			// Base centrale non utilizzata della cavallina
			IF Supporto.Tipologia = CAVALLETTO    THEN
				B := Supporto.YDim - Supporto.DimBaseUtile - Supporto.DimBaseUtile;
				B2 := ( Supporto.YDim / 2 )-supporto.DimBaseUtile ;
				CorYIz := supporto.DimBaseUtile ;
				CorYDe := Supporto.YDim - supporto.DimBaseUtile ;
				BaseAlgulo := ( Supporto.YDim /2) - (Supporto.DimVertice /2)- supporto.DimBaseUtile;
			ELSE
				B := Supporto.YDim - Supporto.DimBaseUtile - Supporto.DimBaseUtile;
				B2 := ( Supporto.YDim / 2 )-supporto.DimBaseUtile ;
			END_IF
			
			//B := Supporto.YDim - Supporto.DimBaseUtile - Supporto.DimBaseUtile;
			//B2 := ( Supporto.YDim / 2 )-supporto.DimBaseUtile ;
			IF (B <= 0 ) THEN
				Errore := ErrBase;
				RETURN;
			END_IF
			
			IF (Supporto.DimBaseUtile <= 0 ) OR (Supporto.DimBaseUtile <= 0 ) THEN
				Errore := ErrLUtile;
			END_IF
			
			b1 := (B - Supporto.DimVertice) / 2;	// base del triangolo rettangolo dell'angolo alfa
			IF (b1 <= 0 ) THEN
				Errore := ErrBaseAlfa;
				RETURN;
			END_IF
			
			h1 := Supporto.HMAX - Supporto.ZDim; // Altezza del triangolo rettangolo dell'angolo alfa
			IF h1 <= 0 THEN
				Errore := ErrAltezzaAlfa;
				RETURN;
			END_IF
			
			(* calcolo angolo alfa dell'inclinazione appoggio della lastra *)
			AngoloAlfa_rad := ATAN( b1 / h1); // Angolo superiore appoggio cavallina (in radianti)
			AlgoloAlfa_gradi := rad_to_deg(AngoloAlfa_rad); 
			
			IF (AlgoloAlfa_gradi >= 90) THEN
				Errore := ErrAngolo;
				RETURN;
			END_IF
			
			(* Calcolo angolo beta dell'eventuale piano di appoggio inclinato della cavallina*)
			AngoloBeta_rad := ATAN( (Supporto.ZDim_Ext1 - Supporto.ZDim) / Supporto.DimBaseUtile); 	// Angolo del piano di appoggio inclinato della cavallina (in radianti)
			AngoloBeta_gradi := rad_to_deg(AngoloBeta_rad);					// Angolo del piano di appoggio inclinato della cavallina (in gradi)
			rad90 := deg_to_rad(90);
			
			IF (AlgoloAlfa_gradi < (AngoloBeta_gradi-1)) AND FALSE (*Quitar alarma pendiente base*) THEN
				Errore := ErrPendenzaBase;					// Angolo alfa deve essere maggiore dell'angolo beta
				RETURN;
			END_IF
			
			// Calcolo lo spessore di ogni singola lastra/falda depositata sul lato della cavallina
			Spessore_Lastra_Inclinata[1] := 0;
			FOR counter2:=2 TO MAXFORMINGSLAB/2 BY 1 DO
				Spessore_Lastra_Inclinata[counter2] := Materiale[TipoElementoDep[counter2-1]].ZDim / COS(AngoloAlfa_rad);
			END_FOR;
			
			// Calcola lo spessore complessivo fino al passo n delle lastre/falde depositate sul singolo lato della cavallina 
			//memset(ADR(Spessore_Lastra_Inclinata_Cumulato), 0 , SIZEOF(Spessore_Lastra_Inclinata_Cumulato));
			
			IF (Spessore_Lastra_Inclinata_Cumulato[2] = 0) THEN
				FOR counter2:=1 TO MAXFORMINGSLAB/2 BY 1 DO
					FOR counter1 := 1 TO counter2 BY 1 DO
						Spessore_Lastra_Inclinata_Cumulato[counter2] := Spessore_Lastra_Inclinata_Cumulato[counter2]+Spessore_Lastra_Inclinata[counter1];
					END_FOR
				END_FOR
			END_IF
			
			// Numero di possibili lastre sul singolo lato
			//FOR counter1:=1 TO MAXFORMINGSLAB/2 BY 1 DO
				//IF (OrdineDeposito[counter1] <> e_Tipo_Elemento_Da_Lavorare.NOT_DEFINED AND OrdineDeposito[counter1] <> TERMINATORE) AND 
				//	((Spessore_Lastra_Inclinata_Cumulato[counter1] >0) AND (Spessore_Lastra_Inclinata_Cumulato[counter1] < Supporto.DimBaseUtile)) THEN
				//		numeroLastre_int := counter1;
				//END_IF
				//IF (OrdineDeposito[counter1] <> e_Tipo_Elemento_Da_Lavorare.NOT_DEFINED AND OrdineDeposito[counter1] <> TERMINATORE) AND 
				//	(Spessore_Lastra_Inclinata_Cumulato[counter1] >= Supporto.DimBaseUtile) THEN
				//		Errore := ErrNumeroPezzi;	// il supervisore mi ha passato troppe lastre rispetto allo spazio utile
				//END_IF
			//END_FOR
			IF (Spessore_Lastra_Inclinata_Cumulato[numeroLastre_int] >= Supporto.DimBaseUtile*2) THEN
				Errore := ErrNumeroPezzi;	// il supervisore mi ha passato troppe lastre rispetto allo spazio utile
			END_IF
			
			// Calcolo lo spostamento del punto centrale e del punto esterno della singola lastra/falda rispetto al punto interno(iniziale) della medesima lastra/falda
			FOR counter2:=1 TO numeroLastre_int BY 1 DO
				Yd1[counter2] := Materiale[TipoElementoDep[counter2]].ZDim / 2 * COS (AngoloAlfa_rad);		// Spostamento Centro lastra da interno lastra in Y
				Zd1[counter2] := Materiale[TipoElementoDep[counter2]].ZDim / 2 * SIN (AngoloAlfa_rad);		// Spostamento Centro lastra da interno lastra in Z
				Yd2[counter2] := Materiale[TipoElementoDep[counter2]].ZDim  * COS (AngoloAlfa_rad);			// Spostamento esterno lastra da interno lastra in Y
				Zd2[counter2] := Materiale[TipoElementoDep[counter2]].ZDim  * SIN (AngoloAlfa_rad);			// Spostamento esterno lastra da interno lastra in Z
			END_FOR
			
			// Calcolo la proiezione mancante di ogni singola lastra/falda; Tramite CI posso calcolare lo spostamento Yd3,Zd3 dovuto al piano inclinato
			// dovuto all'angolo beta. Utilizzo il teorema dei seni per calcolare ogni CI da SLIC
			FOR counter1:=1 TO numeroLastre_int BY 1 DO
				CI[counter1] := (Spessore_Lastra_Inclinata_Cumulato[counter1] * SIN (AngoloBeta_rad) ) / SIN( rad90 + AngoloAlfa_rad - AngoloBeta_rad);
				Yd3[counter1] := -CI[counter1] * SIN(AngoloAlfa_rad);
				Zd3[counter1] := CI[counter1] * COS(AngoloAlfa_rad);
			END_FOR;
			
			// Quota Y e Z del punto di appoggio di ogni lastra sulla cavallina
			// Quota Y e Z del punto interno centrale di ogni lastra; corrisponde a YInternoLastra e ZInternoLastra
			NuPiezasLadoDx := 0 ;
			NuPiezasLadoSx := 0 ;
			FOR counter2:=1 TO numeroLastre_int BY 1 DO
				XInternoLastra[counter2] := Supporto.XDim/2;
				varEven := counter2 MOD 2;
				IF Supporto.Tipologia = CAVALLETTO    THEN
					CASE varEven OF
						0:	
								CASE TipoCalculo OF
								0:
									YCoordinataAppoggioLastra[counter2] := (B/2) + Spessore_Lastra_Inclinata_Cumulato[counter2] + Yd3[counter2];
								
								
								1: 
									NuPiezasLadoDx := NuPiezasLadoDx +1 ;
									YCoordinataAppoggioLastra[counter2] := (CorYDe) + Spessore_Lastra_Inclinata_Cumulato[NuPiezasLadoDx] + Yd3[NuPiezasLadoDx];
									
								END_CASE
						1:
							CASE TipoCalculo OF
								0:
									YCoordinataAppoggioLastra[counter2] := (B/2) + Spessore_Lastra_Inclinata_Cumulato[counter2] - Yd3[counter2];
								
								1:
									NuPiezasLadoSx := NuPiezasLadoSx + 1;
									YCoordinataAppoggioLastra[counter2] := (CorYIz) + Spessore_Lastra_Inclinata_Cumulato[NuPiezasLadoSx] - Yd3[NuPiezasLadoSx];
							END_CASE
					END_CASE
					
					
					ELSE
					YCoordinataAppoggioLastra[counter2] := (B/2) + Spessore_Lastra_Inclinata_Cumulato[counter2] + Yd3[counter2];
						
				END_IF
				//YCoordinataAppoggioLastra[counter2] := (*(B2) +*) Spessore_Lastra_Inclinata_Cumulato[counter2] + Yd3[counter2];
				YInternoLastra[counter2] := YCoordinataAppoggioLastra[counter2] - (Materiale[TipoElementoDep[counter2]].YDim / 2) * SIN (AngoloAlfa_rad);
				ZCoordinataAppoggioLastra[counter2] := Supporto.ZDim + Zd3[counter2];
				ZInternoLastra[counter2] := ZCoordinataAppoggioLastra[counter2] + (Materiale[TipoElementoDep[counter2]].YDim / 2) * COS (AngoloAlfa_rad); 
			END_FOR
	
			(* Calcolo delle coordinate X,Y,Z di ogni singola lastra/falda, centrale o esterno *)
			FOR counter2:=1 TO numeroLastre_int BY 1 DO
				XCentroLastra[counter2] := Supporto.XDim/2;
				YCentroLastra[counter2] := YInternoLastra[counter2] + Yd1[counter2];
				ZCentroLastra[counter2] := ZInternoLastra[counter2] + Zd1[counter2];
				
				XEsternoLastra[counter2] := Supporto.XDim/2;
				YEsternoLastra[counter2] := YInternoLastra[counter2] + Yd2[counter2];	
				ZEsternoLastra[counter2] := ZInternoLastra[counter2] + Zd2[counter2];
			END_FOR;
			
			(* Pulisco le uscite e setto a TERMINATORE tutti gli elementi di FormingSlab*)
			FOR counter1 := 1 TO MAXFORMINGSLAB DO
				FormingSlab.PElement[counter1].Typology := TERMINATORE;
			END_FOR
		//#########################aqui for	
		IF HabiCalTodasCordenadas THEN
				F_ini := 1 ;
				F_Fin := 4 ;
			ELSE
				F_ini := TipoOrdinamento ;
				F_Fin := TipoOrdinamento ;
		END_IF
		FOR CalForCavallete := F_ini TO F_Fin DO
			(* Calcolo delle coordinate X,Y,Z,J del punto finale sulla base del TipoRisultato *)
			CASE CalForCavallete OF
				(* Ordinamento alternato Dx-SX *)	
				1: 
					FOR counter2:=1 TO numeroLastre_int*2 BY 1 DO
						varEven := counter2 MOD 2;	
						CASE varEven OF
							0:	// Lato DX della cavallina
								XFinale[counter2] := Supporto.XDim/2 + Supporto.OFSDE_X180;
								CASE TipoRisultato OF
									1:	
										YFinale[counter2] := -YInternoLastra[(counter2+varEven)/2] + Supporto.OFSDE_Y180;
										ZFinale[counter2] := ZInternoLastra[(counter2+varEven)/2] + Supporto.OFSDE_Z180;
									2:	
										YFinale[counter2] := -YCentroLastra[(counter2+varEven)/2] + Supporto.OFSDE_Y180;
										ZFinale[counter2] := ZCentroLastra[(counter2+varEven)/2] + Supporto.OFSDE_Z180;
									3:	
										YFinale[counter2] := -YEsternoLastra[(counter2+varEven)/2] + Supporto.OFSDE_Y180;
										ZFinale[counter2] := ZEsternoLastra[(counter2+varEven)/2] + Supporto.OFSDE_Z180;
									4:	
										YFinale[counter2] := -YCoordinataAppoggioLastra[(counter2+varEven)/2] + Supporto.OFSDE_Y180;
										ZFinale[counter2] := ZEsternoLastra[(counter2+varEven)/2] + Supporto.OFSDE_Z180;
								END_CASE
								JFinale[counter2] := 180 - AlgoloAlfa_gradi + Supporto.OFSDE_J180; 
							1:	// Lato SX della cavallina
								XFinale[counter2] := Supporto.XDim/2 + Supporto.OFSDE_X0;
								CASE TipoRisultato OF
									1:	
										YFinale[counter2] := YInternoLastra[(counter2+varEven)/2] + Supporto.OFSDE_Y0;
										ZFinale[counter2] := ZInternoLastra[(counter2+varEven)/2] + Supporto.OFSDE_Z0;
									2:	
										YFinale[counter2] := YCentroLastra[(counter2+varEven)/2] + Supporto.OFSDE_Y0;
										ZFinale[counter2] := ZCentroLastra[(counter2+varEven)/2] + Supporto.OFSDE_Z0;
									3:	
										YFinale[counter2] := YEsternoLastra[(counter2+varEven)/2] + Supporto.OFSDE_Y0;
										ZFinale[counter2] := ZEsternoLastra[(counter2+varEven)/2] + Supporto.OFSDE_Z0;
									4:	
										YFinale[counter2] := YCoordinataAppoggioLastra[(counter2+varEven)/2] + Supporto.OFSDE_Y0;
										ZFinale[counter2] := ZEsternoLastra[(counter2+varEven)/2] + Supporto.OFSDE_Z0;
								END_CASE
								JFinale[counter2] := AlgoloAlfa_gradi + Supporto.OFSDE_J0;
						END_CASE
					END_FOR
					
				(* Ordinamento consecutivo prima un lato poi l'altro *)
				2:	
					FOR  CntLados :=  1 TO 2 BY 1 DO
						CASE CntLados OF 
							1:
								FOR counter2 :=1 TO numeroLastre_int BY 1 DO
										CoorFinaleLado_Pri0_Des180[counter2].LadoA.CoordenadaFinale_X := Supporto.XDim/2 + Supporto.OFSDE_X180;
									CASE TipoRisultato OF	
										1:	
											CoorFinaleLado_Pri0_Des180[counter2].LadoA.CoordenadaFinale_Y := YInternoLastra[counter2] + Supporto.OFSDE_Y0;
											CoorFinaleLado_Pri0_Des180[counter2].LadoA.CoordenadaFinale_Z := ZInternoLastra[counter2] + Supporto.OFSDE_Z0;
										2:	
											CoorFinaleLado_Pri0_Des180[counter2].LadoA.CoordenadaFinale_Y := YCentroLastra[counter2] + Supporto.OFSDE_Y0;
											CoorFinaleLado_Pri0_Des180[counter2].LadoA.CoordenadaFinale_Z := ZCentroLastra[counter2] + Supporto.OFSDE_Z0;
										3:	
											CoorFinaleLado_Pri0_Des180[counter2].LadoA.CoordenadaFinale_Y := YEsternoLastra[counter2] + Supporto.OFSDE_Y0;
											CoorFinaleLado_Pri0_Des180[counter2].LadoA.CoordenadaFinale_Z := ZEsternoLastra[counter2] + Supporto.OFSDE_Z0;
										4:	
											CoorFinaleLado_Pri0_Des180[counter2].LadoA.CoordenadaFinale_Y := YCoordinataAppoggioLastra[counter2] + Supporto.OFSDE_Y0;
											CoorFinaleLado_Pri0_Des180[counter2].LadoA.CoordenadaFinale_Z := ZEsternoLastra[counter2] + Supporto.OFSDE_Z0;
									END_CASE
									CoorFinaleLado_Pri0_Des180[counter2].LadoA.CoordenadaFinale_J := AlgoloAlfa_gradi + Supporto.OFSDE_J0;
								END_FOR
								2: 
									FOR counter2:=1 TO numeroLastre_int BY 1 DO
										
										CoorFinaleLado_Pri0_Des180[counter2].LadoA.CoordenadaFinale_X := Supporto.XDim/2 + Supporto.OFSDE_X180;
										CASE TipoRisultato OF
											1:	
												CoorFinaleLado_Pri0_Des180[counter2].LadoB.CoordenadaFinale_Y := -YInternoLastra[counter2] + Supporto.OFSDE_Y180;
												CoorFinaleLado_Pri0_Des180[counter2].LadoB.CoordenadaFinale_Z := ZInternoLastra[counter2] + Supporto.OFSDE_Z180;
											2:	
												CoorFinaleLado_Pri0_Des180[counter2].LadoB.CoordenadaFinale_Y := -YCentroLastra[counter2] + Supporto.OFSDE_Y180;
												CoorFinaleLado_Pri0_Des180[counter2].LadoB.CoordenadaFinale_Z := ZCentroLastra[counter2] + Supporto.OFSDE_Z180;
											3:	
												CoorFinaleLado_Pri0_Des180[counter2].LadoB.CoordenadaFinale_Y := -YEsternoLastra[counter2] + Supporto.OFSDE_Y180;
												//YFinale[counter2] := YCoordinataAppoggioLastra[counter2] ;
												CoorFinaleLado_Pri0_Des180[counter2].LadoB.CoordenadaFinale_Z := ZEsternoLastra[counter2] + Supporto.OFSDE_Z180;
											4:	
												CoorFinaleLado_Pri0_Des180[counter2].LadoB.CoordenadaFinale_Y := -YCoordinataAppoggioLastra[counter2] + Supporto.OFSDE_Y180;
												CoorFinaleLado_Pri0_Des180[counter2].LadoB.CoordenadaFinale_Z := ZEsternoLastra[counter2] + Supporto.OFSDE_Z180;
										END_CASE
										CoorFinaleLado_Pri0_Des180[counter2].LadoB.CoordenadaFinale_J := 180 - AlgoloAlfa_gradi + Supporto.OFSDE_J180; 
									END_FOR
													
							
							END_CASE
						END_FOR
						
							IF NOT HabiCalTodasCordenadas THEN 
								FOR counter2:=1 TO numeroLastre_int BY 1 DO
								IF counter2 <= numeroLastre_int/2 THEN // Lato DX della cavallina
									varEven := counter2 MOD 2;
									XFinale[counter2] := Supporto.XDim/2 + Supporto.OFSDE_X180;
									CASE TipoRisultato OF
										1:	
											YFinale[counter2] := -YInternoLastra[counter2] + Supporto.OFSDE_Y180;
											ZFinale[counter2] := ZInternoLastra[counter2] + Supporto.OFSDE_Z180;
										2:	
											YFinale[counter2] := -YCentroLastra[counter2] + Supporto.OFSDE_Y180;
											ZFinale[counter2] := ZCentroLastra[counter2] + Supporto.OFSDE_Z180;
										3:	
											YFinale[counter2] := -YEsternoLastra[counter2] + Supporto.OFSDE_Y180;
											ZFinale[counter2] := ZEsternoLastra[counter2] + Supporto.OFSDE_Z180;
										4:	
											YFinale[counter2] := -YCoordinataAppoggioLastra[counter2] + Supporto.OFSDE_Y180;
											ZFinale[counter2] :=  ZEsternoLastra[counter2] + Supporto.OFSDE_Z180;
									END_CASE
											JFinale[counter2] := 180 - AlgoloAlfa_gradi + Supporto.OFSDE_J180; 
								ELSE// Lato SX della cavallina
									XFinale[counter2] := Supporto.XDim/2 + Supporto.OFSDE_X0;
									CASE TipoRisultato OF
										1:	
											YFinale[counter2] := YInternoLastra[counter2-numeroLastre_int/2] + Supporto.OFSDE_Y0;
											ZFinale[counter2] := ZInternoLastra[counter2-numeroLastre_int/2] + Supporto.OFSDE_Z0;
										2:	
											YFinale[counter2] := YCentroLastra[counter2-numeroLastre_int/2] + Supporto.OFSDE_Y0;
											ZFinale[counter2] := ZCentroLastra[counter2-numeroLastre_int/2] + Supporto.OFSDE_Z0;
										3:	
											YFinale[counter2] := YEsternoLastra[counter2-numeroLastre_int/2] + Supporto.OFSDE_Y0;
											ZFinale[counter2] := ZEsternoLastra[counter2-numeroLastre_int/2] + Supporto.OFSDE_Z0;
										4:	
											YFinale[counter2] := YCoordinataAppoggioLastra[counter2-numeroLastre_int/2] + Supporto.OFSDE_Y0;
											ZFinale[counter2] := ZEsternoLastra[counter2-numeroLastre_int/2] + Supporto.OFSDE_Z0;
									END_CASE
									JFinale[counter2] := AlgoloAlfa_gradi + Supporto.OFSDE_J0;
								END_IF
							END_FOR
							END_IF
							
				(* Ordinamento consecutivo prima SOLO lato 0° *)
				3:
					FOR counter2:=1 TO numeroLastre_int BY 1 DO
						XFinaleLado_0Grados[counter2] := Supporto.XDim/2 + Supporto.OFSDE_X0;
						CASE TipoRisultato OF
							1:	
								YFinaleLado_0Grados[counter2] := YInternoLastra[counter2-numeroLastre_int/2] + Supporto.OFSDE_Y0;
								ZFinaleLado_0Grados[counter2] := ZInternoLastra[counter2-numeroLastre_int/2] + Supporto.OFSDE_Z0;
							2:	
								YFinaleLado_0Grados[counter2] := YCentroLastra[counter2-numeroLastre_int/2] + Supporto.OFSDE_Y0;
								ZFinaleLado_0Grados[counter2] := ZCentroLastra[counter2-numeroLastre_int/2] + Supporto.OFSDE_Z0;
							3:	
								YFinaleLado_0Grados[counter2] := YEsternoLastra[counter2-numeroLastre_int/2] + Supporto.OFSDE_Y0;
								ZFinaleLado_0Grados[counter2] := ZEsternoLastra[counter2-numeroLastre_int/2] + Supporto.OFSDE_Z0;
							4:	
								YFinaleLado_0Grados[counter2] := YCoordinataAppoggioLastra[counter2-numeroLastre_int/2] + Supporto.OFSDE_Y0;
								ZFinaleLado_0Grados[counter2] := ZEsternoLastra[counter2-numeroLastre_int/2] + Supporto.OFSDE_Z0;
						END_CASE
						JFinaleLado_0Grados[counter2] := AlgoloAlfa_gradi + Supporto.OFSDE_J0;
					END_FOR
					IF NOT HabiCalTodasCordenadas THEN 
						FOR counter2:=1 TO numeroLastre_int BY 1 DO
						XFinale[counter2] := Supporto.XDim/2 + Supporto.OFSDE_X0;
						CASE TipoRisultato OF
							1:	
								YFinale[counter2] := YInternoLastra[counter2-numeroLastre_int/2] + Supporto.OFSDE_Y0;
								ZFinale[counter2] := ZInternoLastra[counter2-numeroLastre_int/2] + Supporto.OFSDE_Z0;
							2:	
								YFinale[counter2] := YCentroLastra[counter2-numeroLastre_int/2] + Supporto.OFSDE_Y0;
								ZFinale[counter2] := ZCentroLastra[counter2-numeroLastre_int/2] + Supporto.OFSDE_Z0;
							3:	
								YFinale[counter2] := YEsternoLastra[counter2-numeroLastre_int/2] + Supporto.OFSDE_Y0;
								ZFinale[counter2] := ZEsternoLastra[counter2-numeroLastre_int/2] + Supporto.OFSDE_Z0;
							4:	
								YFinale[counter2] := YCoordinataAppoggioLastra[counter2-numeroLastre_int/2] + Supporto.OFSDE_Y0;
								ZFinale[counter2] := ZEsternoLastra[counter2-numeroLastre_int/2] + Supporto.OFSDE_Z0;
						END_CASE
						JFinale[counter2] := AlgoloAlfa_gradi + Supporto.OFSDE_J0;
					END_FOR
					END_IF
				(* Ordinamento consecutivo SOLO lato 180 *)
				4:
					FOR counter2:=1 TO numeroLastre_int BY 1 DO
						varEven := counter2 MOD 2;
						XFinaleLado_180Grados[counter2] := Supporto.XDim/2 + Supporto.OFSDE_X180;
						CASE TipoRisultato OF
							1:	
								YFinaleLado_180Grados[counter2] := -YInternoLastra[counter2] + Supporto.OFSDE_Y180;
								ZFinaleLado_180Grados[counter2] := 	ZInternoLastra[counter2] + Supporto.OFSDE_Z180;
							2:	
								YFinaleLado_180Grados[counter2] := -YCentroLastra[counter2] + Supporto.OFSDE_Y180;
								ZFinaleLado_180Grados[counter2] := ZCentroLastra[counter2] + Supporto.OFSDE_Z180;
							3:	
								YFinaleLado_180Grados[counter2] := -YEsternoLastra[counter2] + Supporto.OFSDE_Y180;
								//YFinale[counter2] := YCoordinataAppoggioLastra[counter2] ;
								ZFinaleLado_180Grados[counter2] := ZEsternoLastra[counter2] + Supporto.OFSDE_Z180;
							4:	
								YFinaleLado_180Grados[counter2] := -YCoordinataAppoggioLastra[counter2] + Supporto.OFSDE_Y180;
								ZFinaleLado_180Grados[counter2] := ZEsternoLastra[counter2] + Supporto.OFSDE_Z180;
						END_CASE
						JFinaleLado_180Grados[counter2] := 180 - AlgoloAlfa_gradi + Supporto.OFSDE_J180; 
					END_FOR
					IF NOT HabiCalTodasCordenadas THEN 
						FOR counter2:=1 TO numeroLastre_int BY 1 DO
						varEven := counter2 MOD 2;
						XFinale[counter2] := Supporto.XDim/2 + Supporto.OFSDE_X180;
						CASE TipoRisultato OF
							1:	
								YFinale[counter2] := -YInternoLastra[counter2] + Supporto.OFSDE_Y180;
								ZFinale[counter2] := ZInternoLastra[counter2] + Supporto.OFSDE_Z180;
							2:	
								YFinale[counter2] := -YCentroLastra[counter2] + Supporto.OFSDE_Y180;
								ZFinale[counter2] := ZCentroLastra[counter2] + Supporto.OFSDE_Z180;
							3:	
								YFinale[counter2] := -YEsternoLastra[counter2] + Supporto.OFSDE_Y180;
								//YFinale[counter2] := YCoordinataAppoggioLastra[counter2] ;
								ZFinale[counter2] := ZEsternoLastra[counter2] + Supporto.OFSDE_Z180;
							4:	
								YFinale[counter2] := -YCoordinataAppoggioLastra[counter2] + Supporto.OFSDE_Y180;
								ZFinale[counter2] := ZEsternoLastra[counter2] + Supporto.OFSDE_Z180;
						END_CASE
						JFinale[counter2] := 180 - AlgoloAlfa_gradi + Supporto.OFSDE_J180; 
					END_FOR
					END_IF
		
			5:
					;		
					
					
			END_CASE						
		END_FOR


			
			// Alimentazione della struttura FormingSlab
			FOR counter1:=1 TO MAXFORMINGSLAB DO// numeroLastre_int*2 BY 1 DO
				IF counter1 <= numeroLastre_int THEN
					FormingSlab.Enable := 1;										// Abilitato
					//FormingSlab.Code[1] := 1;
					FormingSlab.PElement[counter1].Typology 			:= OrdineDepositoSxDx[counter1];
					FormingSlab.PElement[counter1].X 					:= XFinale[counter1];
					FormingSlab.PElement[counter1].XDim 				:= Materiale[OrdineDepositoSxDx[counter1]].XDim;		// Dimensione X Lastra
					FormingSlab.PElement[counter1].Y 					:= YFinale[counter1];
					FormingSlab.PElement[counter1].YDim 				:= Materiale[OrdineDepositoSxDx[counter1]].YDim;		// Dimensione Y Lastra
					FormingSlab.PElement[counter1].Z 					:= ZFinale[counter1];
					FormingSlab.PElement[counter1].ZDim 				:= Materiale[OrdineDepositoSxDx[counter1]].ZDim;		// Dimensione Z Lastra
					FormingSlab.PElement[counter1].J 					:= JFinale[counter1];
					FormingSlab.PElement[counter1].CooCavallete 		:= CoorFinaleLado_Pri0_Des180[counter1] ;
				ELSE
					FormingSlab.PElement[counter1].Typology := OrdineDepositoSxDx[counter1];
					FormingSlab.PElement[counter1].X 		:= -1;
					FormingSlab.PElement[counter1].XDim 	:= -1;	
					FormingSlab.PElement[counter1].Y 		:= -1;
					FormingSlab.PElement[counter1].YDim 	:= -1;		
					FormingSlab.PElement[counter1].Z 		:= -1;
					FormingSlab.PElement[counter1].ZDim 	:= -1;	
					FormingSlab.PElement[counter1].J 		:= -1;
				END_IF
			END_FOR		
		

		INCLINATO_LATOSINGOLO:		// Tipo deposito inclinato singolo lato (Bundle)
			numeroLastre_int := 0;
			FOR counter1:=1 TO MAXFORMINGSLAB/2 BY 1 DO
				IF (TipoElementoDep[counter1] > 0) THEN
				numeroLastre_int := numeroLastre_int+1;
				END_IF;
			END_FOR
	
			(* Controlli dati coerenti --- DA FARE --- *)
						
			(* calcolo angolo alfa dell'inclinazione appoggio della lastra *)
			AngoloAlfa_rad := deg_to_rad(Supporto.AngoloAlfaBundle); // Angolo superiore appoggio cavallina (in radianti)
			AlgoloAlfa_gradi := Supporto.AngoloAlfaBundle; 
			
			
			(* Calcolo angolo beta dell'eventuale piano di appoggio inclinato della cavallina*)
			AngoloBeta_rad := AngoloAlfa_rad; 	// Angolo del piano di appoggio inclinato della cavallina (in radianti)
			AngoloBeta_gradi := AlgoloAlfa_gradi;					// Angolo del piano di appoggio inclinato della cavallina (in gradi)
	
			
			// Calcolo lo spessore di ogni singola lastra/falda depositata sul lato della cavallina
			Spessore_Lastra_Inclinata[1] := 0;
			FOR counter2:=2 TO MAXFORMINGSLAB/2 BY 1 DO
				Spessore_Lastra_Inclinata[counter2] := Materiale[TipoElementoDep[counter2-1]].ZDim / COS(AngoloAlfa_rad);
			END_FOR;
			
			// Calcola lo spessore complessivo fino al passo n delle lastre/falde depositate sul singolo lato della cavallina 
			//memset(ADR(Spessore_Lastra_Inclinata_Cumulato), 0 , SIZEOF(Spessore_Lastra_Inclinata_Cumulato));
			
			IF (Spessore_Lastra_Inclinata_Cumulato[2] = 0) THEN
				FOR counter2:=1 TO MAXFORMINGSLAB/2 BY 1 DO
					FOR counter1 := 1 TO counter2 BY 1 DO
						Spessore_Lastra_Inclinata_Cumulato[counter2] := Spessore_Lastra_Inclinata_Cumulato[counter2]+Spessore_Lastra_Inclinata[counter1];
					END_FOR
				END_FOR
			END_IF
			
			// Numero di possibili lastre sul singolo lato
			FOR counter1:=1 TO MAXFORMINGSLAB/2 BY 1 DO
				IF (TipoElementoDep[counter1] > 0) AND ((Spessore_Lastra_Inclinata_Cumulato[counter1] >0) AND (Spessore_Lastra_Inclinata_Cumulato[counter1] < Supporto.DimBaseUtile)) THEN
					numeroLastre_int := counter1;
				END_IF
				IF (Spessore_Lastra_Inclinata_Cumulato[counter1] >= Supporto.DimBaseUtile) THEN
					Errore := ErrNumeroPezzi;	// il supervisore mi ha passato troppe lastre rispetto allo spazio utile
				END_IF
			END_FOR
			
			// Calcolo lo spostamento del punto centrale e del punto esterno della singola lastra/falda rispetto al punto interno(iniziale) della medesima lastra/falda
			FOR counter2:=1 TO numeroLastre_int BY 1 DO
				Yd1[counter2] := Materiale[TipoElementoDep[counter2]].ZDim / 2 * COS (AngoloAlfa_rad);		// Spostamento Centro lastra da interno lastra in Y
				Zd1[counter2] := Materiale[TipoElementoDep[counter2]].ZDim / 2 * SIN (AngoloAlfa_rad);		// Spostamento Centro lastra da interno lastra in Z
				Yd2[counter2] := Materiale[TipoElementoDep[counter2]].ZDim  * COS (AngoloAlfa_rad);			// Spostamento esterno lastra da interno lastra in Y
				Zd2[counter2] := Materiale[TipoElementoDep[counter2]].ZDim  * SIN (AngoloAlfa_rad);			// Spostamento esterno lastra da interno lastra in Z
			END_FOR
			
			// Calcolo la proiezione mancante di ogni singola lastra/falda; Tramite CI posso calcolare lo spostamento Yd3,Zd3 dovuto al piano inclinato
			// dovuto all'angolo beta. Utilizzo il teorema dei seni per calcolare ogni CI da SLIC
			FOR counter1:=1 TO numeroLastre_int BY 1 DO
				CI[counter1] := (Spessore_Lastra_Inclinata_Cumulato[counter1] * SIN (AngoloBeta_rad));
				Yd3[counter1] := -CI[counter1] * SIN(AngoloAlfa_rad);
				Zd3[counter1] := CI[counter1] * COS(AngoloAlfa_rad);
			END_FOR;
			
			// Quota Y e Z del punto di appoggio di ogni lastra sulla cavallina
			// Quota Y e Z del punto interno centrale di ogni lastra; corrisponde a YInternoLastra e ZInternoLastra
			FOR counter2:=1 TO numeroLastre_int BY 1 DO
				XInternoLastra[counter2] := Supporto.XDim/2;
				YCoordinataAppoggioLastra[counter2] := Spessore_Lastra_Inclinata_Cumulato[counter2] + Yd3[counter2];
				YInternoLastra[counter2] := YCoordinataAppoggioLastra[counter2] - (Materiale[TipoElementoDep[counter2]].YDim / 2) * SIN (AngoloAlfa_rad);
				ZCoordinataAppoggioLastra[counter2] := Supporto.ZDim + Zd3[counter2];
				ZInternoLastra[counter2] := ZCoordinataAppoggioLastra[counter2] + (Materiale[TipoElementoDep[counter2]].YDim / 2) * COS (AngoloAlfa_rad); 
			END_FOR
	
			(* Calcolo delle coordinate X,Y,Z di ogni singola lastra/falda, centrale o esterno *)
			FOR counter2:=1 TO numeroLastre_int BY 1 DO
				XCentroLastra[counter2] := Supporto.XDim/2;
				YCentroLastra[counter2] := YInternoLastra[counter2] + Yd1[counter2];
				ZCentroLastra[counter2] := ZInternoLastra[counter2] + Zd1[counter2];
				
				XEsternoLastra[counter2] := Supporto.XDim/2;
				YEsternoLastra[counter2] := YInternoLastra[counter2] + Yd2[counter2];	
				ZEsternoLastra[counter2] := ZInternoLastra[counter2] + Zd2[counter2];
			END_FOR;
			
			(* Pulisco le uscite e setto a TERMINATORE tutti gli elementi di FormingSlab*)
			//memset(ADR(XFinale),0,SIZEOF(XFinale));memset(ADR(YFinale),0,SIZEOF(XFinale));memset(ADR(ZFinale),0,SIZEOF(XFinale));memset(ADR(JFinale),0,SIZEOF(XFinale));
			//memset(ADR(FormingSlab),0,SIZEOF(FormingSlab));
			FOR counter1 := 1 TO MAXFORMINGSLAB DO
				FormingSlab.PElement[counter1].Typology := TERMINATORE;
			END_FOR
			
			(* Calcolo delle coordinate X,Y,Z,J del punto finale sulla base del TipoRisultato *)
			FOR counter2:=1 TO numeroLastre_int BY 1 DO
				CASE supporto.LatoDeposito OF
					180:		// Lato DX della cavallina
						XFinale[counter2] := Supporto.XDim/2 + Supporto.OFSDE_X180;
						CASE TipoRisultato OF
							1:	
								YFinale[counter2] := -YInternoLastra[counter2] + Supporto.OFSDE_Y180;
								ZFinale[counter2] := ZInternoLastra[counter2] + Supporto.OFSDE_Z180;
							2:	
								YFinale[counter2] := -YCentroLastra[counter2] + Supporto.OFSDE_Y180;
								ZFinale[counter2] := ZCentroLastra[counter2] + Supporto.OFSDE_Z180;
							3:	
								YFinale[counter2] := -YEsternoLastra[counter2] + Supporto.OFSDE_Y180;
								ZFinale[counter2] := ZEsternoLastra[counter2] + Supporto.OFSDE_Z180;
						END_CASE
						JFinale[counter2] := 180 - AlgoloAlfa_gradi + Supporto.OFSDE_J180; 
					0:	// Lato SX della cavallina
						XFinale[counter2] := Supporto.XDim/2 + Supporto.OFSDE_X0;
						CASE TipoRisultato OF
							1:	
								YFinale[counter2] := YInternoLastra[counter2] + Supporto.OFSDE_Y0;
								ZFinale[counter2] := ZInternoLastra[counter2] + Supporto.OFSDE_Z0;
							2:	
								YFinale[counter2] := YCentroLastra[counter2] + Supporto.OFSDE_Y0;
								ZFinale[counter2] := ZCentroLastra[counter2] + Supporto.OFSDE_Z0;
							3:	
								YFinale[counter2] := YEsternoLastra[counter2] + Supporto.OFSDE_Y0;
								ZFinale[counter2] := ZEsternoLastra[counter2] + Supporto.OFSDE_Z0;
						END_CASE
						JFinale[counter2] := AlgoloAlfa_gradi + Supporto.OFSDE_J0;
				END_CASE

				
				// Alimentazione della struttura FormingSlab
				FOR counter1:=1 TO numeroLastre_int BY 1 DO
					FormingSlab.Enable := 1;										// Abilitato
					FormingSlab.Code[1] := 1;
					FormingSlab.PElement[counter1].Typology := Materiale[OrdineDepositoSxDx[counter1]].Typology;
					FormingSlab.PElement[counter1].X := XFinale[counter1];
					FormingSlab.PElement[counter1].XDim := Materiale[OrdineDepositoSxDx[counter1]].XDim;		// Dimensione X Lastra
					FormingSlab.PElement[counter1].Y := YFinale[counter1];
					FormingSlab.PElement[counter1].YDim := Materiale[OrdineDepositoSxDx[counter1]].YDim;		// Dimensione Y Lastra
					FormingSlab.PElement[counter1].Z := ZFinale[counter1];
					FormingSlab.PElement[counter1].ZDim := Materiale[OrdineDepositoSxDx[counter1]].ZDim;		// Dimensione Z Lastra
					FormingSlab.PElement[counter1].J := JFinale[counter1];
				END_FOR		
			END_FOR;	
	END_CASE


	// Salvataggio su file della Formatura 
	{region "Salvataggio File Formatura"}
	P_TextModeWrite.database[0,0] := 'X Finale';
	P_TextModeWrite.database[0,1] := 'Y Finale';
	P_TextModeWrite.database[0,2] := 'Z Finale';
	P_TextModeWrite.database[0,3] := 'J Finale';
	CASE TipoDeposito OF
		ORIZZONTALE :	
			P_TextModeWrite.database[0,4] := 'ORIZZONTALE';
			P_TextModeWrite.database[0,5] := UINT_TO_STRING(numeroLastre_int);
		INCLINATO : 
			P_TextModeWrite.database[0,4] := 'INCLINATO';
			P_TextModeWrite.database[0,5] := UINT_TO_STRING(numeroLastre_int*2);
		INCLINATO_LATOSINGOLO :
			P_TextModeWrite.database[0,4] := 'INCLINATO_LATOSINGOLO';
			P_TextModeWrite.database[0,5] := UINT_TO_STRING(numeroLastre_int);	  
	END_CASE
	CASE TipoRisultato OF
		1:	P_TextModeWrite.database[0,6] := 'PUNTO INTERNO';
		2:	P_TextModeWrite.database[0,6] := 'PUNTO CENTRALE';
		3:	P_TextModeWrite.database[0,6] := 'PUNTO ESTERNO';
	END_CASE
	
	FOR counter1 :=1 TO MAXFORMINGSLAB DO
		P_TextModeWrite.database[counter1,0] := LREAL_TO_STRING(XFinale[counter1]);
		P_TextModeWrite.database[counter1,1] := LREAL_TO_STRING(YFinale[counter1]);
		P_TextModeWrite.database[counter1,2] := LREAL_TO_STRING(ZFinale[counter1]);
		P_TextModeWrite.database[counter1,3] := LREAL_TO_STRING(JFinale[counter1]);
	END_FOR
	
	CASE TipoDeposito OF	// Numero di righe da scrivere sul file a seconda che sia CASSA o CAVALLINA
		ORIZZONTALE :	
			P_TextModeWrite.num_Row := numeroLastre_int;
		INCLINATO : 
			P_TextModeWrite.num_Row := numeroLastre_int * 2;
		INCLINATO_LATOSINGOLO : 
			P_TextModeWrite.num_Row := numeroLastre_int;
	END_CASE
	
	{endregion}
	CalcolaFormaturaDone := TRUE;	
	P_TextModeWrite.bWrite := TRUE; //Scrivo log per calcoli
ELSIF NOT CalcolaFormatura AND CalcolaFormaturaDone THEN
	CalcolaFormaturaDone := FALSE;
END_IF

//chiamata fb per log calcoli	
//___________P_TextModeWrite();
IF P_TextModeWrite.bWriteDone AND P_TextModeWrite.bWrite THEN
	P_TextModeWrite.bWrite := FALSE; 
END_IF

END_FUNCTION_BLOCK

// ---- POUs/TFPalletizerData_Lastre/Formatura/FuncionesFormacionParaquitar/Calcolo_Formatura_Completa_Back.TcPOU
FUNCTION_BLOCK Calcolo_Formatura_Completa_Back
VAR_INPUT
	
	Supporto : TFMachinePalletizer_Pallet;
	
	//Materiale : ARRAY [0..MAXTYPE_SLABLAYER] OF Type_SlabLayer;	// Tipo di materiale, Lastra, Falda e dimensioni
	Materiale 		: ARRAY [0..MAXTYPE_SLABLAYER] OF TFMachinePalletizer_PlaceElement;	// Tipo di materiale, Lastra, Falda e dimensioni
	TipoElementoDep 	: ARRAY [1..MAXFORMINGSLAB] OF e_Tipo_Elemento_Da_Lavorare;	// Tipologia del n-esimo elemento di Materiale da depositare (Lstra-falda-terminatore)
	
	TipoRisultato 		: UINT := 3;// Punto utilizzato per coordinate finali di deposito lastra/falda, 1 interno, 2 centro, 3 esterno(default)
	TipoOrdinamento 	: UINT := 1;//Tipologia di ordinamento in deposito 1= alternato (lastra DX-Lastra SX), 2 = consecutivo(prima un lato, poi l'altro lato), 3 = solo lato 0°, 4 = solo lato 180°
	NumeroElementiDaDepositare : UINT;

	PulisciMemoria : BOOL;
	CalcolaFormatura : BOOL;
END_VAR

VAR_OUTPUT
	(* Variabili di uscita della posizione finale del punto di deposito della lastra/falda *)
	XFinale : ARRAY [1..MAXFORMINGSLAB] OF LREAL;		// Coordinata X punto finale n-esima lastra/falda depositata
	YFinale : ARRAY [1..MAXFORMINGSLAB] OF LREAL;		// Coordinata Y punto finale n-esima lastra/falda depositata
	ZFinale : ARRAY [1..MAXFORMINGSLAB] OF LREAL;		// Coordinata Z punto finale n-esima lastra/falda depositata
	JFinale : ARRAY [1..MAXFORMINGSLAB] OF LREAL;		// Coordinata J punto finale n-esima lastra/falda depositata
	
	FormingSlab 			: TFMachinePalletizer_FormingForSlab;
	PulisciMemoriaDone		: BOOL;
	CalcolaFormaturaDone 	: BOOL;
	Errore 					: UINT;
END_VAR
VAR
	TipoDeposito : e_TipologiaDeposito;				// ORIZZONTALE O INCLINATO
	OrdineDepositoSxDx : ARRAY [1..MAXFORMINGSLAB] OF e_Tipo_Elemento_Da_Lavorare;	// Ordine deposito materiale per i due lati, sx e dx (considero di avere il medesimo ordine di deposito dai due lati) (CAVALLINA-INCLINATO)
	
	Spessore_Lastra_Inclinata : ARRAY [1..MAXFORMINGSLAB/2] OF LREAL;				// Occupazione in larghezza della singola lastra (CAVALLINA-INCLINATO)
	Spessore_Lastra_Inclinata_Cumulato : ARRAY [1..MAXFORMINGSLAB/2] OF LREAL;	// Occupazione in larghezza delle nlastre lastre cumulate (CAVALLINA)
	Spessore_Lastra : ARRAY [1..MAXFORMINGSLAB] OF LREAL;							// Occupazione in altezza della singola lastra (CASSA-ORIZZONTALE)
	Spessore_Lastra_Cumulato : ARRAY [1..MAXFORMINGSLAB] OF LREAL;					// Occupazione in altezza delle nlastre lastre cumulate (CASSA-ORIZZONTALE)
	
	YCoordinataAppoggioLastra :  ARRAY [1..MAXFORMINGSLAB/2] OF LREAL;		// Coordinata Y del punto di appoggio della lastra sulla base della cavallina  (CAVALLINA-INCLINATO)
	ZCoordinataAppoggioLastra :  ARRAY [1..MAXFORMINGSLAB/2] OF LREAL;		// Coordinata Z del punto di appoggio della lastra sulla base della cavallina  (CAVALLINA-INCLINATO)
	
	B 	: LREAL;	// Base della cavallina (include i due lati)  (CAVALLINA-INCLINATO)
	B2	: LREAL;	// Base della cavallina (include i due lati)  (CAVALLINA-INCLINATO)
	CorYIz  : LREAL;
	CorYDe : LREAL;
	BaseAlgulo : LREAL ;
	b1 : LREAL;	// base del triangolo rettangolo dell'angolo alfa  (CAVALLINA-INCLINATO)
	h1 : LREAL; // altezza del triangolo rettangolo dell'angolo alfa  (CAVALLINA-INCLINATO)
	Yd1 : ARRAY [1..MAXFORMINGSLAB/2] OF LREAL;	// Spostamento Centro lastra da inizio lastra in Y  (CAVALLINA-INCLINATO)
	Zd1 : ARRAY [1..MAXFORMINGSLAB/2] OF LREAL;	// Spostamento Centro lastra da inizio lastra in Z  (CAVALLINA-INCLINATO)
	Yd2 : ARRAY [1..MAXFORMINGSLAB/2] OF LREAL;	// Spostamento Esterno lastra da inizio lastra in Y  (CAVALLINA-INCLINATO)
	Zd2 : ARRAY [1..MAXFORMINGSLAB/2] OF LREAL;	// Spostamento Esterno lastra da inizio lastra in Z  (CAVALLINA-INCLINATOCAVALLINA)
	Yd3 : ARRAY [1..MAXFORMINGSLAB/2] OF LREAL;	// Spostamento Y dovuto al lato inclinato base appoggio  (CAVALLINA-INCLINATO)
	Zd3 : ARRAY [1..MAXFORMINGSLAB/2] OF LREAL;	// Spostamento Z dovuto al lato inclinato base appoggio  (CAVALLINA-INCLINATO)
	CI : ARRAY [1..MAXFORMINGSLAB/2] OF LREAL;	// Proiezione mancante della lastra dovuta al piano inclinato (CI) - Valorizzata solo se Beta >0  (CAVALLINA-INCLINATO)
	rad90 : LREAL;		// 90° in radianti
	
	(* Angoli piani appoggio lastre, laterale (alfa) e base (beta) cavallina *)
	AngoloAlfa_rad : LREAL;		// Angolo superiore laterale appoggio della lastra (in radianti)  (CAVALLINA-INCLINATO)
	AlgoloAlfa_gradi : LREAL; 	// Angolo superiore laterale appoggio della lastra (in gradi)  (CAVALLINA-INCLINATO)
	AngoloBeta_rad : LREAL;		// Angolo del piano inclinato di appoggio della lastra in radianti  (CAVALLINA-INCLINATO)
	AngoloBeta_gradi : LREAL; 	// Angolo del piano inclinato di appoggio della lastra in gradi  (CAVALLINA-INCLINATO)
	
	QuotaYinizioLastra : ARRAY [1..MAXFORMINGSLAB] OF LREAL;	// Quota Y inizio prima lastra  (CAVALLINA-INCLINATO)
	QuotaZinizioLastra : ARRAY [1..MAXFORMINGSLAB] OF LREAL;	// Quota Z inizio prima lastra  (CAVALLINA-INCLINATO)
	numeroLastre_int : UINT;									// Numero lastre per lato cavallina considerando la dimensione L_Utile1 (int)  (CAVALLINA-CASSA)
	
	(* Variabili di supporto *)
	counter1: UINT := 0;	// contatore per ciclo creazione formatura
	counter2: UINT := 0;	// contatore per ciclo creazione formatura
	varEven : UINT := 0;	// Pari o dispari per lato destro (dispari) o lato sinistro (pari) cavallina
	
	(* Variabili di uscita della posizione del punto interno, centrale ed esterno della lastra *)
	XInternoLastra : ARRAY [1..MAXFORMINGSLAB] OF LREAL;		// Coordinata X punto interno n-esima lastra depositata  (CAVALLINA-CASSA)
	YInternoLastra : ARRAY [1..MAXFORMINGSLAB] OF LREAL;		// Coordinata Y punto interno n-esima lastra depositata  (CAVALLINA-CASSA)
	ZInternoLastra : ARRAY [1..MAXFORMINGSLAB] OF LREAL;		// Coordinata Z punto interno n-esima lastra depositata  (CAVALLINA-CASSA)
	XCentroLastra  : ARRAY [1..MAXFORMINGSLAB] OF LREAL;		// Coordinata X punto centrale n-esima lastra depositata  (CAVALLINA-CASSA)
	YCentroLastra  : ARRAY [1..MAXFORMINGSLAB] OF LREAL;		// Coordinata Y punto centrale n-esima lastra depositata  (CAVALLINA-CASSA)
	ZCentroLastra  : ARRAY [1..MAXFORMINGSLAB] OF LREAL;		// Coordinata Z punto centrale n-esima lastra depositata  (CAVALLINA-CASSA)
	XEsternoLastra : ARRAY [1..MAXFORMINGSLAB] OF LREAL;		// Coordinata X punto esterno n-esima lastra depositata  (CAVALLINA-CASSA)
	YEsternoLastra : ARRAY [1..MAXFORMINGSLAB] OF LREAL;		// Coordinata Y punto esterno n-esima lastra depositata  (CAVALLINA-CASSA)
	ZEsternoLastra : ARRAY [1..MAXFORMINGSLAB] OF LREAL;		// Coordinata Z punto esterno n-esima lastra depositata  (CAVALLINA-CASSA)

	P_TextModeWrite : P_TextModeWrite;
	MemoriaInizializzata : BOOL;
END_VAR

VAR CONSTANT
END_VAR

// Pulisco le variabili interne e le variabili di uscita del FB
IF PulisciMemoria AND NOT PulisciMemoriaDone THEN		// Pulizia delle variabili locali e di uscita
	memset(ADR(XFinale), 0 , SIZEOF(XFinale));memset(ADR(YFinale), 0 , SIZEOF(YFinale));memset(ADR(ZFinale), 0 , SIZEOF(ZFinale));memset(ADR(JFinale), 0 , SIZEOF(JFinale));
	memset(ADR(FormingSlab), 0 , SIZEOF(FormingSlab));
	memset(ADR(Errore), 0 , SIZEOF(Errore));
	memset(ADR(OrdineDepositoSxDx), 0 , SIZEOF(OrdineDepositoSxDx));
	memset(ADR(Spessore_Lastra_Inclinata), 0 , SIZEOF(Spessore_Lastra_Inclinata));memset(ADR(Spessore_Lastra_Inclinata_Cumulato), 0 , SIZEOF(Spessore_Lastra_Inclinata_Cumulato));
	memset(ADR(Spessore_Lastra), 0 , SIZEOF(Spessore_Lastra));memset(ADR(Spessore_Lastra_Cumulato), 0 , SIZEOF(Spessore_Lastra_Cumulato));
	memset(ADR(YCoordinataAppoggioLastra), 0 , SIZEOF(YCoordinataAppoggioLastra));memset(ADR(ZCoordinataAppoggioLastra), 0 , SIZEOF(ZCoordinataAppoggioLastra));
	memset(ADR(B), 0 , SIZEOF(B));memset(ADR(b1), 0 , SIZEOF(b1));memset(ADR(h1), 0 , SIZEOF(h1));
	memset(ADR(Yd1), 0 , SIZEOF(Yd1));memset(ADR(Zd1), 0 , SIZEOF(Zd1));
	memset(ADR(Yd2), 0 , SIZEOF(Yd2));memset(ADR(Zd2), 0 , SIZEOF(Zd2));
	memset(ADR(Yd3), 0 , SIZEOF(Yd3));memset(ADR(Zd3), 0 , SIZEOF(Zd3));
	memset(ADR(CI), 0 , SIZEOF(CI));
	memset(ADR(AngoloAlfa_rad), 0 , SIZEOF(AngoloAlfa_rad));memset(ADR(AngoloBeta_rad), 0 , SIZEOF(AngoloBeta_rad));
	memset(ADR(QuotaYinizioLastra), 0 , SIZEOF(QuotaYinizioLastra));memset(ADR(QuotaZinizioLastra), 0 , SIZEOF(QuotaZinizioLastra));
	memset(ADR(numeroLastre_int), 0 , SIZEOF(numeroLastre_int));
	memset(ADR(XInternoLastra), 0 , SIZEOF(XInternoLastra));memset(ADR(YInternoLastra), 0 , SIZEOF(YInternoLastra));memset(ADR(ZInternoLastra), 0 , SIZEOF(ZInternoLastra));
	memset(ADR(XCentroLastra), 0 , SIZEOF(XCentroLastra));memset(ADR(YCentroLastra), 0 , SIZEOF(YCentroLastra));memset(ADR(ZCentroLastra), 0 , SIZEOF(ZCentroLastra));
	memset(ADR(XEsternoLastra), 0 , SIZEOF(XEsternoLastra));memset(ADR(YEsternoLastra), 0 , SIZEOF(YEsternoLastra));memset(ADR(ZEsternoLastra), 0 , SIZEOF(ZEsternoLastra));
	memset(ADR(Supporto), 0 , SIZEOF(Supporto));
	memset(ADR(Materiale), 0 , SIZEOF(Materiale));
	memset(ADR(TipoElementoDep), 99 , SIZEOF(TipoElementoDep));
	Errore := 0;
	PulisciMemoriaDone := TRUE;
	MemoriaInizializzata := TRUE;
ELSIF NOT PulisciMemoria AND PulisciMemoriaDone THEN
	PulisciMemoriaDone := FALSE;
END_IF

// Calcolo la Formatura, tipo Cassa o Cavallina e salvo su file i risultati ottenuti
IF CalcolaFormatura AND NOT CalcolaFormaturaDone AND MemoriaInizializzata THEN
	// Pulisco le variabili interne e le variabili di uscita del FB
	memset(ADR(XFinale), 0 , SIZEOF(XFinale));memset(ADR(YFinale), 0 , SIZEOF(YFinale));memset(ADR(ZFinale), 0 , SIZEOF(ZFinale));memset(ADR(JFinale), 0 , SIZEOF(JFinale));
	memset(ADR(FormingSlab), 0 , SIZEOF(FormingSlab));
	memset(ADR(Errore), 0 , SIZEOF(Errore));
	memset(ADR(OrdineDepositoSxDx), 0 , SIZEOF(OrdineDepositoSxDx));
	memset(ADR(Spessore_Lastra_Inclinata), 0 , SIZEOF(Spessore_Lastra_Inclinata));memset(ADR(Spessore_Lastra_Inclinata_Cumulato), 0 , SIZEOF(Spessore_Lastra_Inclinata_Cumulato));
	memset(ADR(Spessore_Lastra), 0 , SIZEOF(Spessore_Lastra));memset(ADR(Spessore_Lastra_Cumulato), 0 , SIZEOF(Spessore_Lastra_Cumulato));
	memset(ADR(YCoordinataAppoggioLastra), 0 , SIZEOF(YCoordinataAppoggioLastra));memset(ADR(ZCoordinataAppoggioLastra), 0 , SIZEOF(ZCoordinataAppoggioLastra));
	memset(ADR(B), 0 , SIZEOF(B));memset(ADR(b1), 0 , SIZEOF(b1));memset(ADR(h1), 0 , SIZEOF(h1));
	memset(ADR(Yd1), 0 , SIZEOF(Yd1));memset(ADR(Zd1), 0 , SIZEOF(Zd1));
	memset(ADR(Yd2), 0 , SIZEOF(Yd2));memset(ADR(Zd2), 0 , SIZEOF(Zd2));
	memset(ADR(Yd3), 0 , SIZEOF(Yd3));memset(ADR(Zd3), 0 , SIZEOF(Zd3));
	memset(ADR(CI), 0 , SIZEOF(CI));
	memset(ADR(AngoloAlfa_rad), 0 , SIZEOF(AngoloAlfa_rad));memset(ADR(AngoloBeta_rad), 0 , SIZEOF(AngoloBeta_rad));
	memset(ADR(QuotaYinizioLastra), 0 , SIZEOF(QuotaYinizioLastra));memset(ADR(QuotaZinizioLastra), 0 , SIZEOF(QuotaZinizioLastra));
	memset(ADR(numeroLastre_int), 0 , SIZEOF(numeroLastre_int));
	memset(ADR(XInternoLastra), 0 , SIZEOF(XInternoLastra));memset(ADR(YInternoLastra), 0 , SIZEOF(YInternoLastra));memset(ADR(ZInternoLastra), 0 , SIZEOF(ZInternoLastra));
	memset(ADR(XCentroLastra), 0 , SIZEOF(XCentroLastra));memset(ADR(YCentroLastra), 0 , SIZEOF(YCentroLastra));memset(ADR(ZCentroLastra), 0 , SIZEOF(ZCentroLastra));
	memset(ADR(XEsternoLastra), 0 , SIZEOF(XEsternoLastra));memset(ADR(YEsternoLastra), 0 , SIZEOF(YEsternoLastra));memset(ADR(ZEsternoLastra), 0 , SIZEOF(ZEsternoLastra));

	// Definizione del tipo di deposito a seconda del tipo di supporto utilizzato
	CASE Supporto.Tipologia OF
		PALLET_STANDARD : TipoDeposito := ORIZZONTALE;
		CASSA_STANDARD 	: TipoDeposito := ORIZZONTALE;
		CAVALLETTO 		: TipoDeposito := INCLINATO;
		BUNDLE 			: TipoDeposito := INCLINATO;//INCLINATO_LATOSINGOLO;
	END_CASE
	
	CASE TipoDeposito OF
		ORIZZONTALE:				// Tipo deposito Orizzontale (Cassa o Pallet)
			(* CASO DELLA CASSA/PALLET CON DEPOSITO ORIZZONTALE *)
			
			(* Creo un ordine di deposito generico, per effettuare i test del singolo lato della cavallina, per debug  *)
			numeroLastre_int := 0;
			FOR counter1:=1 TO MAXFORMINGSLAB BY 1 DO
				IF (TipoElementoDep[counter1] <> e_Tipo_Elemento_Da_Lavorare.NOT_DEFINED AND TipoElementoDep[counter1] <> TERMINATORE) THEN
					numeroLastre_int := numeroLastre_int+1;
				END_IF;
			END_FOR
			
			(* Controlli dati coerenti *)
			IF (Supporto.HMAX <= 0 ) 	OR (Supporto.YDim <= 0 ) THEN
				Errore := ErrValori;
			END_IF
			
			IF (Supporto.ZDim <= 0) THEN
				Errore := ErrHBaseInternaNulla;
				RETURN;
			END_IF
			
			IF (Supporto.XDim <= 0) THEN
				Errore := ErroreLBaseNulla;
				RETURN;
			END_IF
			
			FOR counter1 :=1 TO numeroLastre_int DO
				IF (Supporto.YDim+30 <= Materiale[TipoElementoDep[counter1]].YDim) OR (Supporto.XDim+30 <= Materiale[TipoElementoDep[counter1]].XDim) THEN
					Errore := ErrDimensioneCassa;
				RETURN;
				END_IF
			END_FOR
			
			memset(ADR(Spessore_Lastra), 0 , SIZEOF(Spessore_Lastra));
			FOR counter2 := 1 TO MAXFORMINGSLAB BY 1 DO
				Spessore_Lastra[counter2] := Materiale[TipoElementoDep[counter2]].ZDim;
			END_FOR
			
			// Calcola lo spessore complessivo fino al passo n delle lastre/falde depositate sul singolo lato della cavallina 
			memset(ADR(Spessore_Lastra_Cumulato), 0 , SIZEOF(Spessore_Lastra_Cumulato));
			IF (Spessore_Lastra_Cumulato[1] = 0) THEN
				FOR counter2:=1 TO MAXFORMINGSLAB BY 1 DO
					FOR counter1 := 1 TO counter2 BY 1 DO
						Spessore_Lastra_Cumulato[counter2] := Spessore_Lastra_Cumulato[counter2] + Spessore_Lastra[counter1];
					END_FOR
				END_FOR
			END_IF
			
			// Numero di possibili lastre sulla cassa (minore dell'altezza massima)
			FOR counter1:=1 TO MAXFORMINGSLAB BY 1 DO
				IF (TipoElementoDep[counter1] <> e_Tipo_Elemento_Da_Lavorare.NOT_DEFINED AND TipoElementoDep[counter1] <> TERMINATORE) AND ((Spessore_Lastra_Cumulato[counter1] >0) AND 
					(Spessore_Lastra_Cumulato[counter1]+Supporto.ZDim < Supporto.HMAX)) THEN
						numeroLastre_int := counter1;
				END_IF
				IF (Spessore_Lastra_Cumulato[counter1]+Supporto.ZDim >= Supporto.HMAX) AND Supporto.Tipologia <> PALLET_STANDARD AND counter1 <= numeroLastre_int THEN
					Errore := ErrNumeroPezzi;
				END_IF
			END_FOR
			
			// Calcolo il punto Z interno, centrale ed esterno per ogni lastra posizionata sulla cassa
			FOR counter1:=1 TO numeroLastre_int BY 1 DO
				ZInternoLastra[counter1] := Supporto.ZDim + Spessore_Lastra_Cumulato[counter1-1];
				ZCentroLastra[counter1] := Supporto.ZDim + (Spessore_Lastra_Cumulato[counter1-1] + Spessore_Lastra_Cumulato[counter1]) / 2;
				ZEsternoLastra[counter1] := Supporto.ZDim + Spessore_Lastra_Cumulato[counter1];
			END_FOR
			
			(* Pulisco le uscite e setto a TERMINATORE tutti gli elementi di FormingSlab *)
			memset(ADR(XFinale),0,SIZEOF(XFinale));memset(ADR(YFinale),0,SIZEOF(YFinale));memset(ADR(ZFinale),0,SIZEOF(ZFinale));memset(ADR(JFinale),0,SIZEOF(JFinale));
			memset(ADR(FormingSlab),0,SIZEOF(FormingSlab));
			FOR counter1 := 1 TO MAXFORMINGSLAB DO
				FormingSlab.PElement[counter1].Typology := TERMINATORE;
			END_FOR
			
			(* Calcolo delle coordinate X,Y,Z del punto finale sulla base del TipoRisultato *)
			FOR counter2:=1 TO numeroLastre_int BY 1 DO
				XInternoLastra[counter2] := 0; YInternoLastra[counter2] := 0;
				XCentroLastra[counter2] := 0;  YCentroLastra[counter2] := 0;
				XEsternoLastra[counter2] := 0; YEsternoLastra[counter2] := 0;
				
				CASE TipoRisultato OF
					1:	XFinale[counter2] := XInternoLastra[counter2] + Supporto.OFSDE_X90;
						YFinale[counter2] := YInternoLastra[counter2] + Supporto.OFSDE_Y90;
						ZFinale[counter2] := ZInternoLastra[counter2] + Supporto.OFSDE_Z90;
						JFinale[counter2] := 90 + Supporto.OFSDE_J90;
					2:	XFinale[counter2] := XCentroLastra[counter2] + Supporto.OFSDE_X90;
						YFinale[counter2] := YCentroLastra[counter2] + Supporto.OFSDE_Y90;
						ZFinale[counter2] := ZCentroLastra[counter2] + Supporto.OFSDE_Z90;
						JFinale[counter2] := 90  + Supporto.OFSDE_J90;
					3:	XFinale[counter2] := XEsternoLastra[counter2] + Supporto.OFSDE_X90;
						YFinale[counter2] := YEsternoLastra[counter2] + Supporto.OFSDE_Y90;
						ZFinale[counter2] := ZEsternoLastra[counter2] + Supporto.OFSDE_Z90;
						JFinale[counter2] := 90 + Supporto.OFSDE_J90;	
				END_CASE
				
			END_FOR;
			FOR counter1:=1 TO numeroLastre_int BY 1 DO
				FormingSlab.Enable := 1;										// Abilitato
				//FormingSlab.Code[1] := 1;
				//FormingSlab.PElement[counter1].Typology := Materiale[OrdineDeposito[counter1]].Typology;

				//Indico la tipologia di elemnto che vado a depositare in base all'ordine passato dall'esterno
				CASE TipoElementoDep[counter1] OF
					LASTRA:
						FormingSlab.PElement[counter1].Typology := LASTRA;

					FALDA:
						FormingSlab.PElement[counter1].Typology := FALDA;

					TERMINATORE:
						FormingSlab.PElement[counter1].Typology := TERMINATORE;
				
				ELSE
					FormingSlab.PElement[counter1].Typology := e_Tipo_Elemento_Da_Lavorare.NOT_DEFINED;

				END_CASE
				
				FormingSlab.PElement[counter1].XDim := Materiale[TipoElementoDep[counter1]].XDim;		// Dimensione X Lastra		
				FormingSlab.PElement[counter1].YDim := Materiale[TipoElementoDep[counter1]].YDim;		// Dimensione Y Lastra
				FormingSlab.PElement[counter1].ZDim := Materiale[TipoElementoDep[counter1]].ZDim;		// Dimensione Z Lastra
				FormingSlab.PElement[counter1].X := XFinale[counter1];
				FormingSlab.PElement[counter1].Y := YFinale[counter1];
				FormingSlab.PElement[counter1].Z := ZFinale[counter1];
				FormingSlab.PElement[counter1].J := JFinale[counter1];
			END_FOR
		
			
		
		INCLINATO:					// Tipo deposito inclinato ( Cavallina)
			(* CASO DELLA CAVALLINA CON DEPOSITO INCLINATO DAI DUE LATI*)
			
			numeroLastre_int := 0;
			FOR counter1:=1 TO MAXFORMINGSLAB/2 BY 1 DO
				IF (TipoElementoDep[counter1] <> e_Tipo_Elemento_Da_Lavorare.NOT_DEFINED AND TipoElementoDep[counter1] <> TERMINATORE) THEN
					numeroLastre_int := numeroLastre_int+1;
				END_IF;
			END_FOR
	
			(* Replico l'ordine di deposito del singolo lato su entrambi i lati, sx e dx della cavallina *)
			FOR counter1:=1 TO MAXFORMINGSLAB BY 1 DO
				varEven := counter1 MOD 2;
				CASE varEven OF
					0:	
						OrdineDepositoSxDx[counter1] := TipoElementoDep[counter1];//OrdineDeposito[counter1/2];
					1:	
						OrdineDepositoSxDx[counter1] := TipoElementoDep[counter1];//OrdineDeposito[(counter1+varEven)/2];
				END_CASE;
			END_FOR;
			
			(* Controlli dati coerenti *)
			FOR counter1:=1 TO MAXFORMINGSLAB DO
				IF(Materiale[TipoElementoDep[counter1]].XDim <0) OR (Materiale[TipoElementoDep[counter1]].YDim <0) OR 
					(Materiale[TipoElementoDep[counter1]].ZDim <0)  OR (Materiale[TipoElementoDep[counter1]].Typology <0) THEN
						Errore := Errvalori;
						RETURN;
				END_IF
			END_FOR
					
			IF Supporto.ZDim <= 0 THEN//OR (Supporto.ZDim_Int2 <=0) THEN
				Errore := ErrHBaseInternaNulla;
				RETURN;
			END_IF
			
			IF Supporto.ZDim_Ext1 <= 0 AND Supporto.TipoPianoAppoggio = 1 THEN//OR (Supporto.ZDim_Ext2 <=0) THEN
				Errore := ErrHBaseEsternaNulla;
				RETURN;
			END_IF
			
			IF Supporto.ZDim > Supporto.ZDim_Ext1 AND Supporto.TipoPianoAppoggio = 1 THEN//OR (Supporto.ZDim_Int2 > Supporto.ZDim_Ext2) THEN
				Errore := ErrBaseInclinata;
				RETURN;
			END_IF
			
			IF (Supporto.HMAX <= 0) THEN		// altezza cavallina
				Errore := ErrHTotaleNulla;
				RETURN;
			END_IF
			
			IF (Supporto.YDim <= 0) THEN		// larghezza Y cavallina
				Errore := ErroreLBaseNulla;
				RETURN;
			END_IF
			
			// Base centrale non utilizzata della cavallina
			IF Supporto.Tipologia = CAVALLETTO    THEN
				B := Supporto.YDim - Supporto.DimBaseUtile - Supporto.DimBaseUtile;
				B2 := ( Supporto.YDim / 2 )-supporto.DimBaseUtile ;
				CorYIz := supporto.DimBaseUtile ;
				CorYDe := Supporto.YDim - supporto.DimBaseUtile ;
				BaseAlgulo := ( Supporto.YDim /2) - (Supporto.DimVertice /2)- supporto.DimBaseUtile;
			ELSE
				B := Supporto.YDim - Supporto.DimBaseUtile - Supporto.DimBaseUtile;
				B2 := ( Supporto.YDim / 2 )-supporto.DimBaseUtile ;
			END_IF
			
			//B := Supporto.YDim - Supporto.DimBaseUtile - Supporto.DimBaseUtile;
			//B2 := ( Supporto.YDim / 2 )-supporto.DimBaseUtile ;
			IF (B <= 0 ) THEN
				Errore := ErrBase;
				RETURN;
			END_IF
			
			IF (Supporto.DimBaseUtile <= 0 ) OR (Supporto.DimBaseUtile <= 0 ) THEN
				Errore := ErrLUtile;
			END_IF
			
			b1 := (B - Supporto.DimVertice) / 2;	// base del triangolo rettangolo dell'angolo alfa
			IF (b1 <= 0 ) THEN
				Errore := ErrBaseAlfa;
				RETURN;
			END_IF
			
			h1 := Supporto.HMAX - Supporto.ZDim; // Altezza del triangolo rettangolo dell'angolo alfa
			IF h1 <= 0 THEN
				Errore := ErrAltezzaAlfa;
				RETURN;
			END_IF
			
			(* calcolo angolo alfa dell'inclinazione appoggio della lastra *)
			AngoloAlfa_rad := ATAN( b1 / h1); // Angolo superiore appoggio cavallina (in radianti)
			AlgoloAlfa_gradi := rad_to_deg(AngoloAlfa_rad); 
			
			IF (AlgoloAlfa_gradi >= 90) THEN
				Errore := ErrAngolo;
				RETURN;
			END_IF
			
			(* Calcolo angolo beta dell'eventuale piano di appoggio inclinato della cavallina*)
			AngoloBeta_rad := ATAN( (Supporto.ZDim_Ext1 - Supporto.ZDim) / Supporto.DimBaseUtile); 	// Angolo del piano di appoggio inclinato della cavallina (in radianti)
			AngoloBeta_gradi := rad_to_deg(AngoloBeta_rad);					// Angolo del piano di appoggio inclinato della cavallina (in gradi)
			rad90 := deg_to_rad(90);
			
			IF (AlgoloAlfa_gradi < AngoloBeta_gradi) THEN
				Errore := ErrPendenzaBase;					// Angolo alfa deve essere maggiore dell'angolo beta
				RETURN;
			END_IF
			
			// Calcolo lo spessore di ogni singola lastra/falda depositata sul lato della cavallina
			Spessore_Lastra_Inclinata[1] := 0;
			FOR counter2:=2 TO MAXFORMINGSLAB/2 BY 1 DO
				Spessore_Lastra_Inclinata[counter2] := Materiale[TipoElementoDep[counter2-1]].ZDim / COS(AngoloAlfa_rad);
			END_FOR;
			
			// Calcola lo spessore complessivo fino al passo n delle lastre/falde depositate sul singolo lato della cavallina 
			//memset(ADR(Spessore_Lastra_Inclinata_Cumulato), 0 , SIZEOF(Spessore_Lastra_Inclinata_Cumulato));
			
			IF (Spessore_Lastra_Inclinata_Cumulato[2] = 0) THEN
				FOR counter2:=1 TO MAXFORMINGSLAB/2 BY 1 DO
					FOR counter1 := 1 TO counter2 BY 1 DO
						Spessore_Lastra_Inclinata_Cumulato[counter2] := Spessore_Lastra_Inclinata_Cumulato[counter2]+Spessore_Lastra_Inclinata[counter1];
					END_FOR
				END_FOR
			END_IF
			
			// Numero di possibili lastre sul singolo lato
			//FOR counter1:=1 TO MAXFORMINGSLAB/2 BY 1 DO
				//IF (OrdineDeposito[counter1] <> e_Tipo_Elemento_Da_Lavorare.NOT_DEFINED AND OrdineDeposito[counter1] <> TERMINATORE) AND 
				//	((Spessore_Lastra_Inclinata_Cumulato[counter1] >0) AND (Spessore_Lastra_Inclinata_Cumulato[counter1] < Supporto.DimBaseUtile)) THEN
				//		numeroLastre_int := counter1;
				//END_IF
				//IF (OrdineDeposito[counter1] <> e_Tipo_Elemento_Da_Lavorare.NOT_DEFINED AND OrdineDeposito[counter1] <> TERMINATORE) AND 
				//	(Spessore_Lastra_Inclinata_Cumulato[counter1] >= Supporto.DimBaseUtile) THEN
				//		Errore := ErrNumeroPezzi;	// il supervisore mi ha passato troppe lastre rispetto allo spazio utile
				//END_IF
			//END_FOR
			IF (Spessore_Lastra_Inclinata_Cumulato[numeroLastre_int] >= Supporto.DimBaseUtile*2) THEN
				Errore := ErrNumeroPezzi;	// il supervisore mi ha passato troppe lastre rispetto allo spazio utile
			END_IF
			
			// Calcolo lo spostamento del punto centrale e del punto esterno della singola lastra/falda rispetto al punto interno(iniziale) della medesima lastra/falda
			FOR counter2:=1 TO numeroLastre_int BY 1 DO
				Yd1[counter2] := Materiale[TipoElementoDep[counter2]].ZDim / 2 * COS (AngoloAlfa_rad);		// Spostamento Centro lastra da interno lastra in Y
				Zd1[counter2] := Materiale[TipoElementoDep[counter2]].ZDim / 2 * SIN (AngoloAlfa_rad);		// Spostamento Centro lastra da interno lastra in Z
				Yd2[counter2] := Materiale[TipoElementoDep[counter2]].ZDim  * COS (AngoloAlfa_rad);			// Spostamento esterno lastra da interno lastra in Y
				Zd2[counter2] := Materiale[TipoElementoDep[counter2]].ZDim  * SIN (AngoloAlfa_rad);			// Spostamento esterno lastra da interno lastra in Z
			END_FOR
			
			// Calcolo la proiezione mancante di ogni singola lastra/falda; Tramite CI posso calcolare lo spostamento Yd3,Zd3 dovuto al piano inclinato
			// dovuto all'angolo beta. Utilizzo il teorema dei seni per calcolare ogni CI da SLIC
			FOR counter1:=1 TO numeroLastre_int BY 1 DO
				CI[counter1] := (Spessore_Lastra_Inclinata_Cumulato[counter1] * SIN (AngoloBeta_rad) ) / SIN( rad90 + AngoloAlfa_rad - AngoloBeta_rad);
				Yd3[counter1] := -CI[counter1] * SIN(AngoloAlfa_rad);
				Zd3[counter1] := CI[counter1] * COS(AngoloAlfa_rad);
			END_FOR;
			
			// Quota Y e Z del punto di appoggio di ogni lastra sulla cavallina
			// Quota Y e Z del punto interno centrale di ogni lastra; corrisponde a YInternoLastra e ZInternoLastra
			FOR counter2:=1 TO numeroLastre_int BY 1 DO
				XInternoLastra[counter2] := Supporto.XDim/2;
				YCoordinataAppoggioLastra[counter2] := (B/2) + Spessore_Lastra_Inclinata_Cumulato[counter2] + Yd3[counter2];
				//YCoordinataAppoggioLastra[counter2] := (*(B2) +*) Spessore_Lastra_Inclinata_Cumulato[counter2] + Yd3[counter2];
				YInternoLastra[counter2] := YCoordinataAppoggioLastra[counter2] - (Materiale[TipoElementoDep[counter2]].YDim / 2) * SIN (AngoloAlfa_rad);
				ZCoordinataAppoggioLastra[counter2] := Supporto.ZDim + Zd3[counter2];
				ZInternoLastra[counter2] := ZCoordinataAppoggioLastra[counter2] + (Materiale[TipoElementoDep[counter2]].YDim / 2) * COS (AngoloAlfa_rad); 
			END_FOR
	
			(* Calcolo delle coordinate X,Y,Z di ogni singola lastra/falda, centrale o esterno *)
			FOR counter2:=1 TO numeroLastre_int BY 1 DO
				XCentroLastra[counter2] := Supporto.XDim/2;
				YCentroLastra[counter2] := YInternoLastra[counter2] + Yd1[counter2];
				ZCentroLastra[counter2] := ZInternoLastra[counter2] + Zd1[counter2];
				
				XEsternoLastra[counter2] := Supporto.XDim/2;
				YEsternoLastra[counter2] := YInternoLastra[counter2] + Yd2[counter2];	
				ZEsternoLastra[counter2] := ZInternoLastra[counter2] + Zd2[counter2];
			END_FOR;
			
			(* Pulisco le uscite e setto a TERMINATORE tutti gli elementi di FormingSlab*)
			FOR counter1 := 1 TO MAXFORMINGSLAB DO
				FormingSlab.PElement[counter1].Typology := TERMINATORE;
			END_FOR
			
			(* Calcolo delle coordinate X,Y,Z,J del punto finale sulla base del TipoRisultato *)
			CASE TipoOrdinamento OF
				(* Ordinamento alternato Dx-SX *)	
				1: 
					FOR counter2:=1 TO numeroLastre_int*2 BY 1 DO
						varEven := counter2 MOD 2;	
						CASE varEven OF
							0:	// Lato DX della cavallina
								XFinale[counter2] := Supporto.XDim/2 + Supporto.OFSDE_X180;
								CASE TipoRisultato OF
									1:	
										YFinale[counter2] := -YInternoLastra[(counter2+varEven)/2] + Supporto.OFSDE_Y180;
										ZFinale[counter2] := ZInternoLastra[(counter2+varEven)/2] + Supporto.OFSDE_Z180;
									2:	
										YFinale[counter2] := -YCentroLastra[(counter2+varEven)/2] + Supporto.OFSDE_Y180;
										ZFinale[counter2] := ZCentroLastra[(counter2+varEven)/2] + Supporto.OFSDE_Z180;
									3:	
										YFinale[counter2] := -YEsternoLastra[(counter2+varEven)/2] + Supporto.OFSDE_Y180;
										ZFinale[counter2] := ZEsternoLastra[(counter2+varEven)/2] + Supporto.OFSDE_Z180;
								END_CASE
								JFinale[counter2] := 180 - AlgoloAlfa_gradi + Supporto.OFSDE_J180; 
							1:	// Lato SX della cavallina
								XFinale[counter2] := Supporto.XDim/2 + Supporto.OFSDE_X0;
								CASE TipoRisultato OF
									1:	
										YFinale[counter2] := YInternoLastra[(counter2+varEven)/2] + Supporto.OFSDE_Y0;
										ZFinale[counter2] := ZInternoLastra[(counter2+varEven)/2] + Supporto.OFSDE_Z0;
									2:	
										YFinale[counter2] := YCentroLastra[(counter2+varEven)/2] + Supporto.OFSDE_Y0;
										ZFinale[counter2] := ZCentroLastra[(counter2+varEven)/2] + Supporto.OFSDE_Z0;
									3:	
										YFinale[counter2] := YEsternoLastra[(counter2+varEven)/2] + Supporto.OFSDE_Y0;
										ZFinale[counter2] := ZEsternoLastra[(counter2+varEven)/2] + Supporto.OFSDE_Z0;
								END_CASE
								JFinale[counter2] := AlgoloAlfa_gradi + Supporto.OFSDE_J0;
						END_CASE
					END_FOR
					
				(* Ordinamento consecutivo prima un lato poi l'altro *)
				2:
					FOR counter2:=1 TO numeroLastre_int BY 1 DO
						IF counter2 <= numeroLastre_int/2 THEN // Lato DX della cavallina
							varEven := counter2 MOD 2;
							XFinale[counter2] := Supporto.XDim/2 + Supporto.OFSDE_X180;
							CASE TipoRisultato OF
								1:	
									YFinale[counter2] := -YInternoLastra[counter2] + Supporto.OFSDE_Y180;
									ZFinale[counter2] := ZInternoLastra[counter2] + Supporto.OFSDE_Z180;
								2:	
									YFinale[counter2] := -YCentroLastra[counter2] + Supporto.OFSDE_Y180;
									ZFinale[counter2] := ZCentroLastra[counter2] + Supporto.OFSDE_Z180;
								3:	
									YFinale[counter2] := -YEsternoLastra[counter2] + Supporto.OFSDE_Y180;
									ZFinale[counter2] := ZEsternoLastra[counter2] + Supporto.OFSDE_Z180;
							END_CASE
									JFinale[counter2] := 180 - AlgoloAlfa_gradi + Supporto.OFSDE_J180; 
						ELSE// Lato SX della cavallina
							XFinale[counter2] := Supporto.XDim/2 + Supporto.OFSDE_X0;
							CASE TipoRisultato OF
								1:	
									YFinale[counter2] := YInternoLastra[counter2-numeroLastre_int/2] + Supporto.OFSDE_Y0;
									ZFinale[counter2] := ZInternoLastra[counter2-numeroLastre_int/2] + Supporto.OFSDE_Z0;
								2:	
									YFinale[counter2] := YCentroLastra[counter2-numeroLastre_int/2] + Supporto.OFSDE_Y0;
									ZFinale[counter2] := ZCentroLastra[counter2-numeroLastre_int/2] + Supporto.OFSDE_Z0;
								3:	
									YFinale[counter2] := YEsternoLastra[counter2-numeroLastre_int/2] + Supporto.OFSDE_Y0;
									ZFinale[counter2] := ZEsternoLastra[counter2-numeroLastre_int/2] + Supporto.OFSDE_Z0;
							END_CASE
							JFinale[counter2] := AlgoloAlfa_gradi + Supporto.OFSDE_J0;
						END_IF
					END_FOR
				
				(* Ordinamento consecutivo prima SOLO lato 0° *)
				3:
					FOR counter2:=1 TO numeroLastre_int BY 1 DO
						XFinale[counter2] := Supporto.XDim/2 + Supporto.OFSDE_X0;
						CASE TipoRisultato OF
							1:	
								YFinale[counter2] := YInternoLastra[counter2-numeroLastre_int/2] + Supporto.OFSDE_Y0;
								ZFinale[counter2] := ZInternoLastra[counter2-numeroLastre_int/2] + Supporto.OFSDE_Z0;
							2:	
								YFinale[counter2] := YCentroLastra[counter2-numeroLastre_int/2] + Supporto.OFSDE_Y0;
								ZFinale[counter2] := ZCentroLastra[counter2-numeroLastre_int/2] + Supporto.OFSDE_Z0;
							3:	
								YFinale[counter2] := YEsternoLastra[counter2-numeroLastre_int/2] + Supporto.OFSDE_Y0;
								ZFinale[counter2] := ZEsternoLastra[counter2-numeroLastre_int/2] + Supporto.OFSDE_Z0;
						END_CASE
						JFinale[counter2] := AlgoloAlfa_gradi + Supporto.OFSDE_J0;
					END_FOR

				(* Ordinamento consecutivo SOLO lato 180 *)
				4:
					FOR counter2:=1 TO numeroLastre_int BY 1 DO
						varEven := counter2 MOD 2;
						XFinale[counter2] := Supporto.XDim/2 + Supporto.OFSDE_X180;
						CASE TipoRisultato OF
							1:	
								YFinale[counter2] := -YInternoLastra[counter2] + Supporto.OFSDE_Y180;
								ZFinale[counter2] := ZInternoLastra[counter2] + Supporto.OFSDE_Z180;
							2:	
								YFinale[counter2] := -YCentroLastra[counter2] + Supporto.OFSDE_Y180;
								ZFinale[counter2] := ZCentroLastra[counter2] + Supporto.OFSDE_Z180;
							3:	
								YFinale[counter2] := -YEsternoLastra[counter2] + Supporto.OFSDE_Y180;
								//YFinale[counter2] := YCoordinataAppoggioLastra[counter2] ;
								ZFinale[counter2] := ZEsternoLastra[counter2] + Supporto.OFSDE_Z180;
						END_CASE
						JFinale[counter2] := 180 - AlgoloAlfa_gradi + Supporto.OFSDE_J180; 
					END_FOR
			END_CASE						
				
			// Alimentazione della struttura FormingSlab
			FOR counter1:=1 TO MAXFORMINGSLAB DO// numeroLastre_int*2 BY 1 DO
				IF counter1 <= numeroLastre_int THEN
					FormingSlab.Enable := 1;										// Abilitato
					//FormingSlab.Code[1] := 1;
					FormingSlab.PElement[counter1].Typology := OrdineDepositoSxDx[counter1];
					FormingSlab.PElement[counter1].X 		:= XFinale[counter1];
					FormingSlab.PElement[counter1].XDim 	:= Materiale[OrdineDepositoSxDx[counter1]].XDim;		// Dimensione X Lastra
					FormingSlab.PElement[counter1].Y 		:= YFinale[counter1];
					FormingSlab.PElement[counter1].YDim 	:= Materiale[OrdineDepositoSxDx[counter1]].YDim;		// Dimensione Y Lastra
					FormingSlab.PElement[counter1].Z 		:= ZFinale[counter1];
					FormingSlab.PElement[counter1].ZDim 	:= Materiale[OrdineDepositoSxDx[counter1]].ZDim;		// Dimensione Z Lastra
					FormingSlab.PElement[counter1].J 		:= JFinale[counter1];
				ELSE
					FormingSlab.PElement[counter1].Typology := OrdineDepositoSxDx[counter1];
					FormingSlab.PElement[counter1].X 		:= -1;
					FormingSlab.PElement[counter1].XDim 	:= -1;	
					FormingSlab.PElement[counter1].Y 		:= -1;
					FormingSlab.PElement[counter1].YDim 	:= -1;		
					FormingSlab.PElement[counter1].Z 		:= -1;
					FormingSlab.PElement[counter1].ZDim 	:= -1;	
					FormingSlab.PElement[counter1].J 		:= -1;
				END_IF
			END_FOR		
		

		INCLINATO_LATOSINGOLO:		// Tipo deposito inclinato singolo lato (Bundle)
			numeroLastre_int := 0;
			FOR counter1:=1 TO MAXFORMINGSLAB/2 BY 1 DO
				IF (TipoElementoDep[counter1] > 0) THEN
				numeroLastre_int := numeroLastre_int+1;
				END_IF;
			END_FOR
	
			(* Controlli dati coerenti --- DA FARE --- *)
						
			(* calcolo angolo alfa dell'inclinazione appoggio della lastra *)
			AngoloAlfa_rad := deg_to_rad(Supporto.AngoloAlfaBundle); // Angolo superiore appoggio cavallina (in radianti)
			AlgoloAlfa_gradi := Supporto.AngoloAlfaBundle; 
			
			
			(* Calcolo angolo beta dell'eventuale piano di appoggio inclinato della cavallina*)
			AngoloBeta_rad := AngoloAlfa_rad; 	// Angolo del piano di appoggio inclinato della cavallina (in radianti)
			AngoloBeta_gradi := AlgoloAlfa_gradi;					// Angolo del piano di appoggio inclinato della cavallina (in gradi)
	
			
			// Calcolo lo spessore di ogni singola lastra/falda depositata sul lato della cavallina
			Spessore_Lastra_Inclinata[1] := 0;
			FOR counter2:=2 TO MAXFORMINGSLAB/2 BY 1 DO
				Spessore_Lastra_Inclinata[counter2] := Materiale[TipoElementoDep[counter2-1]].ZDim / COS(AngoloAlfa_rad);
			END_FOR;
			
			// Calcola lo spessore complessivo fino al passo n delle lastre/falde depositate sul singolo lato della cavallina 
			//memset(ADR(Spessore_Lastra_Inclinata_Cumulato), 0 , SIZEOF(Spessore_Lastra_Inclinata_Cumulato));
			
			IF (Spessore_Lastra_Inclinata_Cumulato[2] = 0) THEN
				FOR counter2:=1 TO MAXFORMINGSLAB/2 BY 1 DO
					FOR counter1 := 1 TO counter2 BY 1 DO
						Spessore_Lastra_Inclinata_Cumulato[counter2] := Spessore_Lastra_Inclinata_Cumulato[counter2]+Spessore_Lastra_Inclinata[counter1];
					END_FOR
				END_FOR
			END_IF
			
			// Numero di possibili lastre sul singolo lato
			FOR counter1:=1 TO MAXFORMINGSLAB/2 BY 1 DO
				IF (TipoElementoDep[counter1] > 0) AND ((Spessore_Lastra_Inclinata_Cumulato[counter1] >0) AND (Spessore_Lastra_Inclinata_Cumulato[counter1] < Supporto.DimBaseUtile)) THEN
					numeroLastre_int := counter1;
				END_IF
				IF (Spessore_Lastra_Inclinata_Cumulato[counter1] >= Supporto.DimBaseUtile) THEN
					Errore := ErrNumeroPezzi;	// il supervisore mi ha passato troppe lastre rispetto allo spazio utile
				END_IF
			END_FOR
			
			// Calcolo lo spostamento del punto centrale e del punto esterno della singola lastra/falda rispetto al punto interno(iniziale) della medesima lastra/falda
			FOR counter2:=1 TO numeroLastre_int BY 1 DO
				Yd1[counter2] := Materiale[TipoElementoDep[counter2]].ZDim / 2 * COS (AngoloAlfa_rad);		// Spostamento Centro lastra da interno lastra in Y
				Zd1[counter2] := Materiale[TipoElementoDep[counter2]].ZDim / 2 * SIN (AngoloAlfa_rad);		// Spostamento Centro lastra da interno lastra in Z
				Yd2[counter2] := Materiale[TipoElementoDep[counter2]].ZDim  * COS (AngoloAlfa_rad);			// Spostamento esterno lastra da interno lastra in Y
				Zd2[counter2] := Materiale[TipoElementoDep[counter2]].ZDim  * SIN (AngoloAlfa_rad);			// Spostamento esterno lastra da interno lastra in Z
			END_FOR
			
			// Calcolo la proiezione mancante di ogni singola lastra/falda; Tramite CI posso calcolare lo spostamento Yd3,Zd3 dovuto al piano inclinato
			// dovuto all'angolo beta. Utilizzo il teorema dei seni per calcolare ogni CI da SLIC
			FOR counter1:=1 TO numeroLastre_int BY 1 DO
				CI[counter1] := (Spessore_Lastra_Inclinata_Cumulato[counter1] * SIN (AngoloBeta_rad));
				Yd3[counter1] := -CI[counter1] * SIN(AngoloAlfa_rad);
				Zd3[counter1] := CI[counter1] * COS(AngoloAlfa_rad);
			END_FOR;
			
			// Quota Y e Z del punto di appoggio di ogni lastra sulla cavallina
			// Quota Y e Z del punto interno centrale di ogni lastra; corrisponde a YInternoLastra e ZInternoLastra
			FOR counter2:=1 TO numeroLastre_int BY 1 DO
				XInternoLastra[counter2] := Supporto.XDim/2;
				YCoordinataAppoggioLastra[counter2] := Spessore_Lastra_Inclinata_Cumulato[counter2] + Yd3[counter2];
				YInternoLastra[counter2] := YCoordinataAppoggioLastra[counter2] - (Materiale[TipoElementoDep[counter2]].YDim / 2) * SIN (AngoloAlfa_rad);
				ZCoordinataAppoggioLastra[counter2] := Supporto.ZDim + Zd3[counter2];
				ZInternoLastra[counter2] := ZCoordinataAppoggioLastra[counter2] + (Materiale[TipoElementoDep[counter2]].YDim / 2) * COS (AngoloAlfa_rad); 
			END_FOR
	
			(* Calcolo delle coordinate X,Y,Z di ogni singola lastra/falda, centrale o esterno *)
			FOR counter2:=1 TO numeroLastre_int BY 1 DO
				XCentroLastra[counter2] := Supporto.XDim/2;
				YCentroLastra[counter2] := YInternoLastra[counter2] + Yd1[counter2];
				ZCentroLastra[counter2] := ZInternoLastra[counter2] + Zd1[counter2];
				
				XEsternoLastra[counter2] := Supporto.XDim/2;
				YEsternoLastra[counter2] := YInternoLastra[counter2] + Yd2[counter2];	
				ZEsternoLastra[counter2] := ZInternoLastra[counter2] + Zd2[counter2];
			END_FOR;
			
			(* Pulisco le uscite e setto a TERMINATORE tutti gli elementi di FormingSlab*)
			//memset(ADR(XFinale),0,SIZEOF(XFinale));memset(ADR(YFinale),0,SIZEOF(XFinale));memset(ADR(ZFinale),0,SIZEOF(XFinale));memset(ADR(JFinale),0,SIZEOF(XFinale));
			//memset(ADR(FormingSlab),0,SIZEOF(FormingSlab));
			FOR counter1 := 1 TO MAXFORMINGSLAB DO
				FormingSlab.PElement[counter1].Typology := TERMINATORE;
			END_FOR
			
			(* Calcolo delle coordinate X,Y,Z,J del punto finale sulla base del TipoRisultato *)
			FOR counter2:=1 TO numeroLastre_int BY 1 DO
				CASE supporto.LatoDeposito OF
					180:		// Lato DX della cavallina
						XFinale[counter2] := Supporto.XDim/2 + Supporto.OFSDE_X180;
						CASE TipoRisultato OF
							1:	
								YFinale[counter2] := -YInternoLastra[counter2] + Supporto.OFSDE_Y180;
								ZFinale[counter2] := ZInternoLastra[counter2] + Supporto.OFSDE_Z180;
							2:	
								YFinale[counter2] := -YCentroLastra[counter2] + Supporto.OFSDE_Y180;
								ZFinale[counter2] := ZCentroLastra[counter2] + Supporto.OFSDE_Z180;
							3:	
								YFinale[counter2] := -YEsternoLastra[counter2] + Supporto.OFSDE_Y180;
								ZFinale[counter2] := ZEsternoLastra[counter2] + Supporto.OFSDE_Z180;
						END_CASE
						JFinale[counter2] := 180 - AlgoloAlfa_gradi + Supporto.OFSDE_J180; 
					0:	// Lato SX della cavallina
						XFinale[counter2] := Supporto.XDim/2 + Supporto.OFSDE_X0;
						CASE TipoRisultato OF
							1:	
								YFinale[counter2] := YInternoLastra[counter2] + Supporto.OFSDE_Y0;
								ZFinale[counter2] := ZInternoLastra[counter2] + Supporto.OFSDE_Z0;
							2:	
								YFinale[counter2] := YCentroLastra[counter2] + Supporto.OFSDE_Y0;
								ZFinale[counter2] := ZCentroLastra[counter2] + Supporto.OFSDE_Z0;
							3:	
								YFinale[counter2] := YEsternoLastra[counter2] + Supporto.OFSDE_Y0;
								ZFinale[counter2] := ZEsternoLastra[counter2] + Supporto.OFSDE_Z0;
						END_CASE
						JFinale[counter2] := AlgoloAlfa_gradi + Supporto.OFSDE_J0;
				END_CASE

				
				// Alimentazione della struttura FormingSlab
				FOR counter1:=1 TO numeroLastre_int BY 1 DO
					FormingSlab.Enable := 1;										// Abilitato
					FormingSlab.Code[1] := 1;
					FormingSlab.PElement[counter1].Typology := Materiale[OrdineDepositoSxDx[counter1]].Typology;
					FormingSlab.PElement[counter1].X := XFinale[counter1];
					FormingSlab.PElement[counter1].XDim := Materiale[OrdineDepositoSxDx[counter1]].XDim;		// Dimensione X Lastra
					FormingSlab.PElement[counter1].Y := YFinale[counter1];
					FormingSlab.PElement[counter1].YDim := Materiale[OrdineDepositoSxDx[counter1]].YDim;		// Dimensione Y Lastra
					FormingSlab.PElement[counter1].Z := ZFinale[counter1];
					FormingSlab.PElement[counter1].ZDim := Materiale[OrdineDepositoSxDx[counter1]].ZDim;		// Dimensione Z Lastra
					FormingSlab.PElement[counter1].J := JFinale[counter1];
				END_FOR		
			END_FOR;	
	END_CASE


	// Salvataggio su file della Formatura 
	{region "Salvataggio File Formatura"}
	P_TextModeWrite.database[0,0] := 'X Finale';
	P_TextModeWrite.database[0,1] := 'Y Finale';
	P_TextModeWrite.database[0,2] := 'Z Finale';
	P_TextModeWrite.database[0,3] := 'J Finale';
	CASE TipoDeposito OF
		ORIZZONTALE :	
			P_TextModeWrite.database[0,4] := 'ORIZZONTALE';
			P_TextModeWrite.database[0,5] := UINT_TO_STRING(numeroLastre_int);
		INCLINATO : 
			P_TextModeWrite.database[0,4] := 'INCLINATO';
			P_TextModeWrite.database[0,5] := UINT_TO_STRING(numeroLastre_int*2);
		INCLINATO_LATOSINGOLO :
			P_TextModeWrite.database[0,4] := 'INCLINATO_LATOSINGOLO';
			P_TextModeWrite.database[0,5] := UINT_TO_STRING(numeroLastre_int);	  
	END_CASE
	CASE TipoRisultato OF
		1:	P_TextModeWrite.database[0,6] := 'PUNTO INTERNO';
		2:	P_TextModeWrite.database[0,6] := 'PUNTO CENTRALE';
		3:	P_TextModeWrite.database[0,6] := 'PUNTO ESTERNO';
	END_CASE
	
	FOR counter1 :=1 TO MAXFORMINGSLAB DO
		P_TextModeWrite.database[counter1,0] := LREAL_TO_STRING(XFinale[counter1]);
		P_TextModeWrite.database[counter1,1] := LREAL_TO_STRING(YFinale[counter1]);
		P_TextModeWrite.database[counter1,2] := LREAL_TO_STRING(ZFinale[counter1]);
		P_TextModeWrite.database[counter1,3] := LREAL_TO_STRING(JFinale[counter1]);
	END_FOR
	
	CASE TipoDeposito OF	// Numero di righe da scrivere sul file a seconda che sia CASSA o CAVALLINA
		ORIZZONTALE :	
			P_TextModeWrite.num_Row := numeroLastre_int;
		INCLINATO : 
			P_TextModeWrite.num_Row := numeroLastre_int * 2;
		INCLINATO_LATOSINGOLO : 
			P_TextModeWrite.num_Row := numeroLastre_int;
	END_CASE
	
	{endregion}
	CalcolaFormaturaDone := TRUE;	
	P_TextModeWrite.bWrite := TRUE; //Scrivo log per calcoli
ELSIF NOT CalcolaFormatura AND CalcolaFormaturaDone THEN
	CalcolaFormaturaDone := FALSE;
END_IF

//chiamata fb per log calcoli	
//  P_TextModeWrite();
IF P_TextModeWrite.bWriteDone AND P_TextModeWrite.bWrite THEN
	P_TextModeWrite.bWrite := FALSE; 
END_IF

END_FUNCTION_BLOCK

// ---- POUs/TFPalletizerData_Lastre/Formatura/Utility/CSV read_write in text mode/P_TextModeRead.TcPOU
(* Reading of CSV file in text mode. None of the field value is containing any non-printing control characters like line feed, carriage return, quotation marks, semicolon... *)
FUNCTION_BLOCK P_TextModeRead
VAR_INPUT
	leggi		: BOOL;
	bRead		: BOOL := FALSE;(* Rising edge starts program execution *)
	sFileName	: T_MaxString := 'C:\CSVData\TextModeGenRead.csv';(* CSV source file path and name *)
END_VAR

VAR_OUTPUT
	bReadDone : BOOL := FALSE;
END_VAR

VAR
	sNetId			: T_AmsNetId := '';	(* TwinCAT system network address *)
	sCSVLine		: T_MaxString := '';(* Single CSV text line (row, record), we are using string as record buffer (your are able to see read fields)  *)
	sCSVField		: T_MaxString := '';(* Single CSV field value (column, record field) *)
	bBusy			: BOOL;
	bError			: BOOL;
	nErrId			: UDINT;
	nRow	 		: UDINT 	:= 0;(* Row number (record) *)
	nColumn			: UDINT 	:= 0;(* Column number (record field) *)
	hFile			: UINT		:= 0;(* File handle of the source file *)
	step			: DWORD 	:= 0;
	fbFileOpen		: FB_FileOpen;(* Opens file *)
	fbFileClose		: FB_FileClose;(* Closes file *)
	fbFileGets		: FB_FileGets;(* Reads one record (line) *)
	fbReader		: FB_CSVMemBufferReader;(* Helper function block used to parse CSV data bytes (single record line) *)

	database		: ARRAY[0..MAX_CSV_ROWS, 0..MAX_CSV_COLUMNS ] OF STRING(MAX_CSV_FIELD_LENGTH);(* Target PLC database *)
END_VAR

IF bRead = TRUE THEN
	bReadDone := FALSE;		// Inizio un nuovo ciclo di lettura
END_IF


CASE step OF
	0:	(* Wait for rising edge at bRead variable *)
		IF bRead THEN
			bRead	:= FALSE;
			bBusy 	:= TRUE;
			bError	:= FALSE;
			nErrId	:= 0;
			hFile	:= 0;
			nRow	:= 0;
			nColumn	:= 0;
			MEMSET( ADR( database ), 0, SIZEOF( database ) );
			step 		:= 1;
		END_IF

	1:	(* Open source file *)
		fbFileOpen(  bExecute := FALSE  );
		fbFileOpen( sNetId := sNetId, sPathName := sFileName, nMode := FOPEN_MODEREAD OR FOPEN_MODETEXT,(* Open file in TEXT mode! *)
					ePath := PATH_GENERIC, bExecute := TRUE );
		step := 2;

	2:(* Wait until open not busy *)
		fbFileOpen( bExecute := FALSE, bError => bError, nErrID => nErrID, hFile => hFile );
		IF NOT fbFileOpen.bBusy THEN
			IF NOT fbFileOpen.bError THEN
				step := 3;
			ELSE(* Error: file not found? *)
				step := 100;
			END_IF
		END_IF

	3:	(* Read single line (record) *)
		fbFileGets( bExecute := FALSE );
		fbFileGets( sNetId := sNetId, hFile := hFile, bExecute := TRUE );
		step := 4;

	4:(* Wait until read not busy *)
		fbFileGets( bExecute := FALSE, bError => bError, nErrID => nErrID, sLine => sCSVLine );
		IF NOT fbFileGets.bBusy THEN
			IF NOT fbFileGets.bError THEN
				IF fbFileGets.bEOF THEN
					step := 10;(* End of file reached => Close source file *)
				ELSE

					(* FB_FileGets returns text line without the CR (carriage return) character.
					We have to restore the CR character (replace the $L character with $R$L characters) *)
					IF RIGHT( sCSVLine, 1 ) = '$L' THEN
						sCSVLine := REPLACE( sCSVLine, '$R$L', 2, LEN( sCSVLine ) );
					END_IF

					step := 5;
				END_IF
			ELSE(* Error *)
				step := 100;
			END_IF
		END_IF

	5:(* Parse single line (record) *)
		fbReader.eCmd := eEnumCmd_First;(* Read first field value *)
		REPEAT
			fbReader( pBuffer := ADR( sCSVLine ), cbBuffer := SIZEOF( sCSVLine ), getValue => sCSVField );
			IF fbReader.bOk THEN
				fbReader.eCmd := eEnumCmd_Next;(* Read next field value *)

				IF ( nRow <= MAX_CSV_ROWS ) THEN
					IF ( nColumn <= MAX_CSV_COLUMNS ) THEN
						database[nRow, nColumn] := CSVFIELD_TO_STRING( sCSVField, FALSE );(* TODO: Save or use the field value in your application *)
					END_IF
				END_IF

				nColumn := nColumn + 1;(* Increment number of read columns *)
				IF fbReader.bCRLF THEN(* CRLF == TRUE => End of reacord reached *)
					nRow 		:= nRow + 1;(* Increment number of read records *)
					nColumn 	:= 0;(* Reset number of columns *)
				END_IF

			ELSE(* Error: End of record reached or all fields read *)
				step := 3;(* Try to read next line *)
			END_IF
		UNTIL NOT fbReader.bOk
		END_REPEAT

	10:	(* Close source file *)
		fbFileClose( bExecute := FALSE );
		fbFileClose( sNetId := sNetId, hFile := hFile, bExecute := TRUE );
		step := 11;

	11:(* Wait until close not busy *)
		fbFileClose( bExecute := FALSE, bError => bError, nErrID => nErrID );
		IF ( NOT fbFileClose.bBusy ) THEN
			hFile := 0;
			step := 100;
		END_IF

	100: (* Error or ready step => cleanup *)
		IF ( hFile <> 0 ) THEN
			step := 10; (* Close the source file *)
		ELSE
			bBusy := FALSE;
			bReadDone := TRUE;
			step := 0;	(* Ready *)
		END_IF

END_CASE

END_FUNCTION_BLOCK

// ---- POUs/TFPalletizerData_Lastre/TFPalletizerPackValidationSlab.TcPOU
FUNCTION TFPalletizerPackValidationSlab : UINT
VAR_INPUT
	WorkArea : TFMachinePalletizer_WorkArea;
	WorkAreaState : TFMachinePalletizer_WorkAreaState;
	WorkPickPointState : POINTER TO ARRAY [1..MAXPICKPOINT] OF TFMachinePalletizer_WorkPickPoint_State;
	Forming : POINTER TO ARRAY [1..MAXFORMING] OF TFMachinePalletizer_FormingForSlab;
	PickPoint : UINT;
END_VAR
VAR
	wpp : UINT;
	i : INT;
	PackOffset : REAL;
	CodeAssignedToWA : BOOL; // TRUE se i codice è assegnato ad almeno una WA
	fcode : INT;
END_VAR

TFPalletizerPackValidationSlab := 0; 
PackOffset := 50.0;
wpp:=PickPoint;
//FOR wpp:=1 TO MAXPICKPOINT DO
	(* Verifico disponibilità Pacco *)
	IF WorkPickPointState^[wpp].ProdPresence = WORKPICKPOINT_PRODOTTO_PRESENTE THEN
		fcode := TFPalletizerGetFormingFromCodeSlab(Forming,WorkPickPointState^[wpp].Code);
		IF fcode = 0 THEN
			TFPalletizerPackValidationSlab := ErrPACKCODENOTVALID; // Codice non associato a formatura
			RETURN;			
		ELSIF (WorkPickPointState^[wpp].Element.XDim < Forming^[fcode].PElement[WorkAreaState.P].XDim - PackOffset OR
				WorkPickPointState^[wpp].Element.XDim > Forming^[fcode].PElement[WorkAreaState.P].XDim + PackOffset) OR
				(WorkPickPointState^[wpp].Element.YDim < Forming^[fcode].PElement[WorkAreaState.P].YDim - PackOffset  OR
				WorkPickPointState^[wpp].Element.YDim > Forming^[fcode].PElement[WorkAreaState.P].YDim + PackOffset) OR
				(WorkPickPointState^[wpp].Element.ZDim < Forming^[fcode].PElement[WorkAreaState.P].ZDim - PackOffset OR
				WorkPickPointState^[wpp].Element.ZDim > Forming^[fcode].PElement[WorkAreaState.P].ZDim+ PackOffset)THEN
					TFPalletizerPackValidationSlab := ErrPACKDIMENSIONNOTVALID; // Grandezze pacco errate
					RETURN;
			END_IF	
	END_IF
//END_FOR	

TFPalletizerPackValidationSlab := 0;

END_FUNCTION

// ---- POUs/TFPalletizerData_Lastre/TFPalletizerPickRollerPriority.TcPOU
FUNCTION TFPalletizerPickRollerPriority : uINT (*Restituisce il numero del Pick-Point Sul quale deve può essere effettuato il prelievo*)
VAR_INPUT
	WorkArea 					: POINTER TO ARRAY [1..MAXAREA] OF TFMachinePalletizer_WorkArea;
	WorkAreaState 				: POINTER TO ARRAY [1..MAXAREA] OF TFMachinePalletizer_WorkAreaState;
	LastRequetsID : string;	(* Codice univoco ultimo prodotto scaricato *)
	Abilita_Priorita_Impostata_Da_Rulliere : BOOL;	(* Se TRUE la priorità del prelievo è gestita della rulliere *)
	//Priorita_Avanzata_Abilitata	: BOOL;					(* Se TRUE la priorità del prelievo è gestita in modo ottimale, 
	//												 	cerco di completare la postazione più completa *) 		
	
END_VAR
VAR
	wpp : UINT;
	pc : INT;
	WPP_Ordinati_Per_Priorita : ARRAY[1..MAXAREA] OF UINT;
	Indice_WPP_Ordinati : ARRAY[1..MAXAREA] OF UINT;
	Indice_Tmp : UINT;
	i	: UINT;
END_VAR

(* Ordinamento in ordine decrescente di Priorità.. in questo modo si cerca la disponibilità sulla rulliera con priorià più alta *)
IF Abilita_Priorita_Impostata_Da_Rulliere THEN
	FOR i := 1 TO MAXAREAPRESENT DO
		WPP_Ordinati_Per_Priorita[i] := INT_TO_UINT(WorkAreaState^[i].TransportState.Priority);
		Indice_WPP_Ordinati[i] := i;
	END_FOR	
	FOR wpp:= 1 TO MAXAREAPRESENT DO 
		IF WPP_Ordinati_Per_Priorita[wpp] <= WPP_Ordinati_Per_Priorita[wpp+1] THEN
			Indice_Tmp := Indice_WPP_Ordinati[wpp];
			Indice_WPP_Ordinati[wpp] := wpp + 1;
 			Indice_WPP_Ordinati[wpp+1] := Indice_Tmp;
			wpp := 1;
		END_IF
	END_FOR
END_IF
(* Per tutte le WorkPickPoint Attive *)
FOR wpp := 1 TO MAXAREAPRESENT DO
	IF WorkArea^[Indice_WPP_Ordinati[wpp]].Enable = 1 THEN
		(* Verifico disponibilità Lastra *)
		IF WorkAreaState^[Indice_WPP_Ordinati[wpp]].TransportState.State = WORKPICKPOINT_STATE_AUTO THEN
			IF WorkAreaState^[Indice_WPP_Ordinati[wpp]].TransportState.ProdPresence = WORKPICKPOINT_PRODOTTO_PRESENTE THEN
				(* Verifico se il codice è giusto *)
				IF WorkAreaState^[Indice_WPP_Ordinati[wpp]].TransportState.DataElement.WorkingID = LastRequetsID AND LastRequetsID <> '' THEN
					TFPalletizerPickRollerPriority := (Indice_WPP_Ordinati[wpp]);
					RETURN;
				ELSE
					;//Proseguo
				END_IF
			END_IF
		END_IF
	END_IF
END_FOR
TFPalletizerPickRollerPriority := 1;//Nel caso non abbia trovato nulla metto la postazione 1 come postazione di Default

END_FUNCTION

// ---- POUs/TFPalletizerData_Lastre/TFPalletizerGetNumPickPointForLayerCode.TcPOU
(* Restituisce il numero del Pick-Point in cui è presente LA FALDA col codice desiderato, se restituisce -1, nessun Pick-Point ha il codice *)
FUNCTION TFPalletizerGetNumPickPointForLayerCode : UINT 
VAR_INPUT
	WorkPickPoint : POINTER TO ARRAY [1..MAXPICKPOINT] OF TFMachinePalletizer_WorkPickPointSlab;
	WorkPickPointState : POINTER TO ARRAY [1..MAXPICKPOINT] OF TFMachinePalletizer_WorkPickPoint_State;
	LayerCode : INT;
END_VAR
VAR
	pickpoint : UINT;
END_VAR

(* Restituisce il numero del Pick-Point in cui è presente LA FALDA col codice desiderato, se restituisce -1, nessun Pick-Point ha il codice *)
(* Per tutti i Pick-Point *)
FOR pickpoint:=1 TO MAXPICKPOINT DO
	(* Se il Pick Point è Abilitato *)
	IF WorkPickPoint^[pickpoint].Enable = 1 THEN
		(* Se il Pick Point è di tipo Magazzino Falde *)
		IF WorkPickPoint^[pickpoint].Tipologia = MAGAZZINO_FALDE THEN
			(* Se è presente almeno una falda *)
			IF WorkPickPointState^[WorkPickPoint^[pickpoint].ID].ProdPresence = PROD_PRESENTE THEN
				(* Se il codice coincide con quello richiesto *)
				IF WorkPickPointState^[WorkPickPoint^[pickpoint].ID].Code = LayerCode THEN
					(* La funzione restituisce il numero del Pick-Point *)
					TFPalletizerGetNumPickPointForLayerCode := (pickpoint);
					RETURN;
				END_IF	
			END_IF				
		END_IF
	END_IF
END_FOR
TFPalletizerGetNumPickPointForLayerCode := 0;

END_FUNCTION

// ---- POUs/TFPalletizerData_Lastre/TFPalletizerGetWPPFromLastraCode.TcPOU
FUNCTION TFPalletizerGetWPPFromLastraCode : UINT (*Restituisce il numero della WorkArea sulla quale c'è la priorità maggiore per il prelievo, se stessa priorità si da in ordine crescente*)
VAR_INPUT
	WorkPickPoint : POINTER TO ARRAY [1..MAXPICKPOINT] OF TFMachinePalletizer_WorkPickPointSlab;
	WorkPickPointState : POINTER TO ARRAY [1..MAXPICKPOINT] OF TFMachinePalletizer_WorkPickPoint_State;
	PCode : INT;	(* Codice della postazione sulla quale si vorrebbe fare il deposito *)
	Abilita_Priorita_Impostata_Da_Rulliere : BOOL;	(* Se TRUE la priorità del prelievo è gestita della rulliere *)
	//Priorita_Avanzata_Abilitata	: BOOL;					(* Se TRUE la priorità del prelievo è gestita in modo ottimale, 
	//												 	cerco di completare la postazione più completa *) 		
END_VAR
VAR
	wpp : UINT;
	pc : INT;
	WPP_Ordinati_Per_Priorita : ARRAY[1..MAXPICKPOINT] OF UINT;
	Indice_WPP_Ordinati : ARRAY[1..MAXPICKPOINT] OF UINT;
	Indice_Tmp : UINT;
	i	: UINT;
END_VAR

(* Ordinamento in ordine decrescente di Priorità.. in questo modo si cerca la disponibilità sulla rulliera con priorià più alta *)
(*IF Abilita_Priorita_Impostata_Da_Rulliere THEN
	FOR i := 1 TO MAXPICKPOINT DO
		WPP_Ordinati_Per_Priorita[i] := INT_TO_UINT(WorkPickPointState^[wpp].Priority);
		Indice_WPP_Ordinati[i] := i;
	END_FOR	
	FOR wpp:= 1 TO MAXPICKPOINT DO 
		IF WPP_Ordinati_Per_Priorita[wpp] <= WPP_Ordinati_Per_Priorita[wpp+1] THEN
			Indice_Tmp := Indice_WPP_Ordinati[wpp];
			Indice_WPP_Ordinati[wpp] := wpp + 1;
 			Indice_WPP_Ordinati[wpp+1] := Indice_Tmp;
			wpp := 1;
		END_IF
	END_FOR
END_IF*)
(* Per tutte le WorkPickPoint Attive *)
FOR wpp := 1 TO MAXPICKPOINT DO
	IF WorkPickPoint^[wpp].Enable = 1 THEN
		(* Verifico disponibilità Lastra *)
		IF WorkPickPointState^[wpp].State = WORKPICKPOINT_STATE_AUTO THEN
			IF WorkPickPointState^[wpp].ProdPresence = WORKPICKPOINT_PRODOTTO_PRESENTE THEN
				(* Verifico se il codice è giusto *)
				IF WorkPickPointState^[wpp].Code = PCode THEN
					TFPalletizerGetWPPFromLastraCode := (wpp);
					RETURN;
				END_IF
			END_IF
		END_IF
	END_IF
END_FOR
TFPalletizerGetWPPFromLastraCode := 0;

END_FUNCTION

// ---- POUs/TFPrograms/TFUps.TcPOU
PROGRAM TFUps
VAR
END_VAR

(* call UPS-FB instance in first lines of the fastest PLC Task *)
fbUPS(eUpsMode := eUpsMode);
(* eUpsMode =							in case of powerfailure:
	 eSUPS_WrPersistData_Shutdown 		writing of persistent data + shutdown
	 eSUPS_WrPersistData_NoShutdown 	writing of PERSISTENT data, no shutdown
	 eSUPS_CheckPowerStatus 			reports powerfailure without ACTION (no writing, no shutdown) 
	 eSUPS_ImmediateShutdown 			skips writing of data, immediate shutdown
*)

(* evaluate UPS State *)
IF eGlobalSUpsState = eSUPS_PowerFailure THEN
	(* first cycle of powerfailure *)
	(* execute code that should only be done once with each powerfailure, i.e. increase powerfailure counter *)
	iPowerFailureCounter := iPowerFailureCounter + 1;
ELSIF eGlobalSUpsState > eSUPS_PowerFailure THEN
	(* next cycles of powerfailure *)
	(* skip regular code execution for the remaining cycles of the powerfailure/writing of persistent data/quick shutdown  ... *)
	RETURN;
END_IF

iPowerCounter := iPowerCounter + 1;

END_PROGRAM

// ---- GlobalTextList.TcGTLO
TEXTLIST GlobalTextList
  54 = '%1.1f'
  55 = '%3.1f'
  172 = '%5.1f'
  0 = '%5.3f'
  171 = '%5.f'
  32 = '%d'
  33 = '%f'
  238 = '%I'
  239 = '%i'
  35 = '%s'
  659 = '0°'
  904 = '180°'
  411 = '90°'
  151 = 'aaa'
  243 = 'ABILITAZIONE CICLO A STEP'
  1598 = 'Abilitazione tastori emergenza'
  241 = 'ABILITAZIONE TEST'
  260 = 'ABILITAZIONE TEST SENZA AUX'
  18 = 'Acceleration'
  14 = 'ActPosition'
  161 = 'Actual Torque %'
  169 = 'Actual Torque (Lib) %'
  168 = 'Actual Torque From DRIVE %*10'
  166 = 'Actual Torque To DRIVE %*10'
  15 = 'ActVelocity'
  231 = 'ADD PACK'
  651 = 'APRI F 1'
  814 = 'APRI F 2'
  967 = 'APRI L 1'
  471 = 'APRI L2'
  147 = 'ate'
  409 = 'ATTIVA NUOVO ORDINE'
  56 = 'Auto'
  83 = 'Automatic'
  177 = 'Ax1'
  180 = 'Ax10'
  207 = 'Ax12'
  208 = 'Ax13'
  211 = 'Ax14'
  178 = 'Ax2'
  203 = 'Ax3'
  206 = 'Ax4'
  201 = 'Ax5'
  202 = 'Ax6'
  196 = 'Ax7'
  195 = 'Ax8'
  179 = 'Ax9'
  217 = 'Backward'
  2650 = 'BLOCCO'
  458 = 'CALIBRAZIONE OVEM'
  40 = 'Case'
  210 = 'CHAIN DOWN'
  209 = 'CHAIN UP'
  427 = 'CHIUDI F 1'
  419 = 'CHIUDI F 2'
  447 = 'CHIUDI L 1'
  968 = 'CHIUDI L 2'
  262 = 'CICLO A STEP OFF'
  261 = 'CICLO A STEP ON'
  251 = 'CICLO DEPOSITO FALDA'
  256 = 'CICLO DEPOSITO PACCO'
  254 = 'CICLO DEPOSITO PALLET'
  237 = 'CICLO DI FALDA'
  234 = 'CICLO DI RIPOSO'
  236 = 'CICLO PALLET'
  250 = 'Ciclo Prelievo Falda'
  252 = 'CICLO PRELIEVO FALDA'
  255 = 'CICLO PRELIEVO PACCO'
  253 = 'CICLO PRELIEVO PALLET'
  1813 = 'Ciclo Senza Aspirazione'
  182 = 'Cmd'
  39 = 'Cmd Exe'
  38 = 'Cmd Exe Case'
  123 = 'Code'
  110 = 'Command'
  37 = 'Command Exe'
  222 = 'Coupler Close'
  220 = 'Coupler Down'
  221 = 'Coupler Opern'
  219 = 'Coupler Up'
  230 = 'CYCLE LAYER'
  229 = 'CYCLE PALLET'
  19 = 'Deceleration'
  20 = 'Distance'
  41 = 'DO'
  119 = 'Emergency'
  120 = 'Enable'
  198 = 'Entrance ok'
  200 = 'ENTRANCENO'
  199 = 'ENTRANCEOK'
  34 = 'Error'
  53 = 'Error Extra'
  911 = 'Errore Attivazione Formatura'
  187 = 'exit ok'
  193 = 'EXITNO'
  190 = 'ExitOk'
  192 = 'EXITOK'
  302 = 'Falda'
  452 = 'FALDA\nOFF'
  450 = 'FALDA \nON'
  92 = 'FAST'
  144 = 'Forming - F'
  216 = 'Forward'
  99 = 'Gate\nAccess 1'
  100 = 'Gate\nAccess 2'
  98 = 'Gate Access 1'
  259 = 'Gestione Assi'
  124 = 'H'
  13 = 'HALT'
  104 = 'Handling'
  146 = 'HANDLING'
  10 = 'HOME'
  9 = 'HOME+'
  113 = 'ID'
  2278 = 'ID Lastra'
  2270 = 'ID Supporto'
  28 = 'J'
  57 = 'Jog'
  4 = 'JOG +'
  5 = 'JOG -'
  16 = 'JOG+'
  17 = 'JOG-'
  130 = 'Jolly'
  69 = 'JPick'
  226 = 'Jpick'
  227 = 'JPlace'
  29 = 'K'
  70 = 'KPick'
  228 = 'Kpick'
  74 = 'KPickMode'
  73 = 'KPickTorque'
  88 = 'KPickType'
  89 = 'KPlaceMode'
  58 = 'Layer'
  145 = 'Layer - L'
  127 = 'DoLearn_Z'
  126 = 'Learn_Z'
  142 = 'LGV Footprint'
  141 = 'LGV LetIn'
  140 = 'LGV Req'
  49 = 'LOAD'
  175 = 'Load'
  165 = 'Load Torque %'
  181 = 'LOAD/UNLOAD'
  112 = 'm'
  30 = 'MAchine'
  47 = 'Machine'
  80 = 'MAn/Auto'
  81 = 'Man/Auto'
  82 = 'Manual'
  164 = 'Max Torque %'
  77 = 'Mission'
  61 = 'Mission state'
  62 = 'Mission State'
  111 = 'mm'
  76 = 'Mode'
  214 = 'Morsa aperta'
  215 = 'Morsa chiusa'
  21 = 'MOVE'
  24 = 'Move\nAbolute'
  25 = 'Move\nAbsolute'
  23 = 'Move Ab\nolute'
  22 = 'Move Absolute'
  102 = 'MovePathInkeId'
  103 = 'MovePathInvokeId'
  101 = 'MovePathVelo'
  407 = 'Numero'
  2262 = 'N° Lastre'
  60 = 'Pack'
  143 = 'Pack - P'
  59 = 'Pallet'
  31 = 'Palletizer'
  154 = 'PathSegmentID'
  153 = 'PathVelo'
  51 = 'PICK'
  78 = 'Pick'
  1138 = 'PINZA'
  52 = 'PLACE'
  79 = 'Place'
  152 = 'PN'
  147 = 'Pos/Neg'
  146 = 'Pos/Neg - PN'
  1 = 'Position'
  242 = 'POTENZA'
  7 = 'Power'
  8 = 'POWER'
  118 = 'Power\nOFF'
  117 = 'Power\nON'
  116 = 'Power\nON/OFF'
  184 = 'POWER OF'
  185 = 'POWER OFF'
  183 = 'POWER ON'
  115 = 'Power ON/OFF'
  6 = 'Power+'
  63 = 'PPick'
  65 = 'PPlace'
  48 = 'PRELOAD'
  163 = 'Product On Gripper'
  186 = 'PX Presence'
  205 = 'PXClose'
  194 = 'PXDown'
  191 = 'PXExit'
  218 = 'PXHOME'
  204 = 'PXOpen'
  188 = 'PXPresence'
  189 = 'PXpresence'
  197 = 'PXUp'
  11 = 'RESET'
  87 = 'Reset'
  449 = 'RESET ERRORI FORMATURA'
  428 = 'Richiesta nuovo Work Order '
  2301 = 'Riposo'
  46 = 'Robot'
  90 = 'ROBOT'
  2398 = 'SBLOCCO'
  162 = 'Set Torque %'
  170 = 'Set Torque (Lib) %'
  167 = 'Set Torque To DRIVE %*10'
  128 = 'Slow'
  114 = 'SSDO'
  85 = 'Start'
  105 = 'START'
  91 = 'Start\nReset'
  144 = 'START   RESET'
  143 = 'START RESET'
  145 = 'START/RESET'
  36 = 'State'
  263 = 'Stati Missione'
  2254 = 'Stato'
  257 = 'STATO MISSIONE'
  258 = 'STATO W.A.M'
  84 = 'Step'
  235 = 'STEP CICLO'
  12 = 'STOP'
  86 = 'Stop'
  224 = 'Stop Down'
  223 = 'Stop Up'
  158 = 'Strapper 1'
  160 = 'Strapper 2'
  159 = 'Strapper2'
  93 = 'SUCTION'
  97 = 'SUCTION\nDOWN'
  95 = 'SUCTION\nOFF'
  94 = 'SUCTION\nON'
  96 = 'SUCTION\nUP'
  129 = 'Taped'
  240 = 'TEST_ENABLE'
  213 = 'Tilter DOWN'
  212 = 'Tilter UP'
  121 = 'Tipology'
  75 = 'Torque'
  173 = 'Torque %'
  174 = 'Torque Position'
  64 = 'TPick'
  106 = 'Transport 1'
  153 = 'Transport 10'
  154 = 'Transport 11'
  155 = 'Transport 12'
  156 = 'Transport 13'
  232 = 'Transport 13A'
  233 = 'Transport 13B'
  157 = 'Transport 14'
  107 = 'Transport 2'
  108 = 'Transport 3'
  109 = 'Transport 4'
  148 = 'Transport 5'
  149 = 'Transport 6'
  150 = 'Transport 7'
  151 = 'Transport 8'
  152 = 'Transport 9'
  122 = 'Typology'
  125 = 'Typoloy'
  50 = 'UNLOAD'
  176 = 'Unload'
  3 = 'Velocity'
  42 = 'WF0'
  43 = 'WF0 Case'
  44 = 'WF1 Case'
  45 = 'WF2 Case'
  244 = 'WF3 Case'
  245 = 'WF4 Case'
  246 = 'WF5 Case'
  247 = 'WF6 Case'
  248 = 'WF7 Case'
  249 = 'WF8 Case'
  647 = 'Work Order Attuale'
  365 = 'Work Order Richiesto'
  131 = 'WorkArea'
  2 = 'X'
  66 = 'XPick'
  26 = 'Y'
  67 = 'YPick'
  27 = 'Z'
  68 = 'ZPick'
  72 = 'ZPickMode'
  71 = 'ZPickTorque'
  132 = '[1]'
  133 = '[2]'
  134 = '[3]'
  135 = '[4]'
  136 = '[5]'
  137 = '[6]'
  138 = '[7]'
  139 = '[8]'
  225 = '[9]'
END_TEXTLIST

// ---- POUs/TFVisuText/HandlingModulesCmd.TcTLO
TEXTLIST HandlingModulesCmd
  0 = 'NOP'
  10 = 'STOP'
  20 = 'RESET'
  60 = 'POWER'
  100 = 'HOME'
  300 = 'MAN'
  500 = 'LOAD'
  3000 = 'MOVE'
  800 = 'UNLOAD'
  1000 = 'DO'
   = ''
END_TEXTLIST

// ---- POUs/TFVisuText/HandlingModulesState.TcTLO
TEXTLIST HandlingModulesState
  10 = 'Stop Run'
  19 = 'Stop End'
  20 = 'Reset Run'
  21 = 'Reset End'
  60 = 'Power Run'
  69 = 'Power End'
  100 = 'Home Run'
  109 = 'Home End'
  300 = 'Man Run'
  399 = 'Man End'
  500 = 'Load Run'
  599 = 'Load End'
  3000 = 'Move Run'
  3099 = 'Move End'
  800 = 'Unload Run'
  899 = 'Unload End'
  1000 = 'Do Run'
  1099 = 'Do End'
  1 = ''
   = ''
END_TEXTLIST

// ---- POUs/TFVisuText/KPickMode.TcTLO
TEXTLIST KPickMode
  0 = 'Suction'
  1 = 'Position'
  2 = 'Position+Torque'
   = ''
END_TEXTLIST

// ---- POUs/TFVisuText/KUnLoadMode.TcTLO
TEXTLIST KUnLoadMode
  0 = 'Suction'
  1 = 'Position'
   = ''
END_TEXTLIST

// ---- POUs/TFVisuText/KPickType.TcTLO
TEXTLIST KPickType
  0 = 'Pack'
  1 = 'Pallet'
  2 = 'Layer'
   = ''
END_TEXTLIST

// ---- POUs/TFVisuText/KLoadMode.TcTLO
TEXTLIST KLoadMode
  0 = 'Suction'
  1 = 'Position'
  2 = 'Position+Torque'
   = ''
END_TEXTLIST

// ---- POUs/TFVisuText/KProduct.TcTLO
TEXTLIST KProduct
  0 = 'Loading'
  1 = 'Loaded'
  2 = 'Unloading'
  3 = 'Unloaded'
   = ''
END_TEXTLIST

// ---- POUs/TFVisuText/KPlaceMode.TcTLO
TEXTLIST KPlaceMode
  0 = 'Suction'
  1 = 'Position'
   = ''
END_TEXTLIST

// ---- POUs/TFVisuText/MissionText.TcTLO
TEXTLIST MissionText
  0 = 'No Operation'
  1 = 'Init'
  2 = 'Picking...'
  3 = 'Picked'
  4 = 'Loading...'
  5 = 'Loaded'
  6 = 'Placing...'
  7 = 'Placed'
  8 = 'Unloading...'
  9 = 'Unloaded'
  10 = 'End'
  99 = 'Error'
   = ''
END_TEXTLIST

// ---- POUs/TFVisuText/PXExitYesNo.TcTLO
TEXTLIST PXExitYesNo
  FALSE = 'NO'
  TRUE = 'YES'
   = ''
END_TEXTLIST

// ---- POUs/TFVisuText/WorkAreaLearn.TcTLO
TEXTLIST WorkAreaLearn
  0 = 'Disabled'
  1 = 'Enabled (ToBe)'
  2 = 'Enabled (Done)'
   = ''
END_TEXTLIST

// ---- POUs/TFVisuText/WorkAreaLGVLetIn.TcTLO
TEXTLIST WorkAreaLGVLetIn
  0 = 'Nop'
  1 = 'LGV Req In'
  2 = 'LGV End'
   = ''
END_TEXTLIST

// ---- POUs/TFVisuText/WorkAreaLGVReq.TcTLO
TEXTLIST WorkAreaLGVReq
  0 = 'Nop'
  1 = 'LGV Request'
  2 = 'LGV Ok In'
   = ''
END_TEXTLIST

// ---- POUs/TFVisuText/WorkAreaStatePN.TcTLO
TEXTLIST WorkAreaStatePN
  0 = 'Positive'
  1 = 'Negative'
   = ''
END_TEXTLIST

// ---- POUs/TFVisuText/WorkAreaTypology.TcTLO
TEXTLIST WorkAreaTypology
  0 = '-'
  1 = 'Pallet (Magazine)'
  2 = 'Pallet (Work)'
  3 = 'Layer (Magazine)'
   = ''
END_TEXTLIST

// ---- POUs/TFVisuText/WorkAreaYesNo.TcTLO
TEXTLIST WorkAreaYesNo
  0 = 'No'
  1 = 'Yes'
   = ''
END_TEXTLIST

// ---- POUs/TFVisuText/WorkAreaState.TcTLO
TEXTLIST WorkAreaState
  0 = 'F+D'
  1 = 'O+D'
  2 = 'F+Wg'
  3 = 'O+Wg'
  4 = 'O+Wd'
  5 = 'O+Wd+D'
  6 = 'O+Tg'
  7 = 'O+Tg+D'
  8 = 'O+Td'
  9 = 'O+Td+D'
  10 = 'O+E'
  11 = 'O+E+D'
  12 = 'O+Lr'
  13 = 'O+Lr+D'
  14 = 'O+Li'
  15 = 'O+Li+D'
  16 = 'O+Le'
  17 = 'O+Le+D'
   = ''
END_TEXTLIST

